LIN {X 0,Y 208.823,Z 674.449,A -85,B 0,C 180,E1 -21153.863,E2 -21153.863} C_VEL
LIN {X 0,Y 207.998,Z 678.952,A -85,B 0,C 180,E1 -21156.795,E2 -21156.795} C_VEL
LIN {X 0,Y 207.528,Z 682.383,A -85,B 0,C 180,E1 -21159.752,E2 -21159.752} C_VEL
LIN {X 0,Y 207.417,Z 684.105,A -85,B 0,C 180,E1 -21161.733,E2 -21161.733} C_VEL
LIN {X 0,Y 207.417,Z 685.435,A -85,B 0,C 180,E1 -21163.724,E2 -21163.724} C_VEL
LIN {X 0,Y 207.605,Z 686.333,A -85,B 0,C 180,E1 -21165.716,E2 -21165.716} C_VEL
LIN {X 0,Y 208.504,Z 686.886,A -85,B 0,C 180,E1 -21169.702,E2 -21169.702} C_VEL
LIN {X 0,Y 209.212,Z 686.573,A -85,B 0,C 180,E1 -21171.689,E2 -21171.689} C_VEL
LIN {X 0,Y 210.098,Z 685.804,A -85,B 0,C 180,E1 -21173.67,E2 -21173.67} C_VEL
LIN {X 0,Y 211.584,Z 684.174,A -85,B 0,C 180,E1 -21176.257,E2 -21176.257} C_VEL
LIN {X 0,Y 213.864,Z 680.916,A -85,B 0,C 180,E1 -21179.537,E2 -21179.537} C_VEL
LIN {X 0,Y 216.359,Z 676.881,A -85,B 0,C 180,E1 -21182.377,E2 -21182.377} C_VEL
LIN {X 0,Y 219.278,Z 671.481,A -85,B 0,C 180,E1 -21185.237,E2 -21185.237} C_VEL
LIN {X 0,Y 222.734,Z 664.359,A -85,B 0,C 180,E1 -21188.121,E2 -21188.121} C_VEL
LIN {X 0,Y 226.294,Z 656.011,A -85,B 0,C 180,E1 -21190.711,E2 -21190.711} C_VEL
LIN {X 0,Y 229.453,Z 647.343,A -85,B 0,C 180,E1 -21192.851,E2 -21192.851} C_VEL
LIN {X 0,Y 232.75,Z 636.876,A -85,B 0,C 180,E1 -21194.899,E2 -21194.899} C_VEL
LIN {X 0,Y 235.49,Z 626.613,A -85,B 0,C 180,E1 -21196.459,E2 -21196.459} C_VEL
LIN {X 0,Y 237.985,Z 614.319,A -85,B 0,C 180,E1 -21197.929,E2 -21197.929} C_VEL
LIN {X 0,Y 238.322,Z 612.312,A -85,B 0,C 180,E1 -21198.142,E2 -21198.142} C_VEL
LIN {X 0,Y 233.556,Z 615.33,A -85,B 0,C 180,E1 -21198.792,E2 -21198.792} C_VEL
LIN {X 0,Y 232.873,Z 615.574,A -85,B 0,C 180,E1 -21198.917,E2 -21198.917} C_VEL
LIN {X 0,Y 228.743,Z 619.885,A -85,B 0,C 180,E1 -21199.24,E2 -21199.24} C_VEL
LIN {X 0,Y 225.248,Z 622.285,A -85,B 0,C 180,E1 -21199.699,E2 -21199.699} C_VEL
LIN {X 0,Y 223.173,Z 622.996,A -85,B 0,C 180,E1 -21200.11,E2 -21200.11} C_VEL
LIN {X 0,Y 220.737,Z 624.617,A -85,B 0,C 180,E1 -21200.449,E2 -21200.449} C_VEL
LIN {X 0,Y 218.711,Z 626.309,A -85,B 0,C 180,E1 -21200.666,E2 -21200.666} C_VEL
LIN {X 0,Y 217.399,Z 627.014,A -85,B 0,C 180,E1 -21200.888,E2 -21200.888} C_VEL
LIN {X 0,Y 215.398,Z 627.078,A -85,B 0,C 180,E1 -21201.466,E2 -21201.466} C_VEL
LIN {X 0,Y 214.764,Z 627.721,A -85,B 0,C 180,E1 -21201.855,E2 -21201.855} C_VEL
LIN {X 0,Y 214.34,Z 629.899,A -85,B 0,C 180,E1 -21202.213,E2 -21202.213} C_VEL
LIN {X 0,Y 213.369,Z 648.073,A -85,B 0,C 180,E1 -21203.272,E2 -21203.272} C_VEL
LIN {X 0,Y 212.299,Z 661.771,A -85,B 0,C 180,E1 -21204.452,E2 -21204.452} C_VEL
LIN {X 0,Y 211.049,Z 675.35,A -85,B 0,C 180,E1 -21206.054,E2 -21206.054} C_VEL
LIN {X 0,Y 209.703,Z 687.117,A -85,B 0,C 180,E1 -21207.858,E2 -21207.858} C_VEL
LIN {X 0,Y 208.34,Z 699.065,A -85,B 0,C 180,E1 -21210.162,E2 -21210.162} C_VEL
LIN {X 0,Y 207.069,Z 709.634,A -85,B 0,C 180,E1 -21212.73,E2 -21212.73} C_VEL
LIN {X 0,Y 206.085,Z 718.236,A -85,B 0,C 180,E1 -21215.308,E2 -21215.308} C_VEL
LIN {X 0,Y 205.251,Z 726.508,A -85,B 0,C 180,E1 -21218.403,E2 -21218.403} C_VEL
LIN {X 0,Y 204.782,Z 732.079,A -85,B 0,C 180,E1 -21220.973,E2 -21220.973} C_VEL
LIN {X 0,Y 204.444,Z 737.792,A -85,B 0,C 180,E1 -21224.276,E2 -21224.276} C_VEL
LIN {X 0,Y 204.435,Z 741.499,A -85,B 0,C 180,E1 -21227.089,E2 -21227.089} C_VEL
LIN {X 0,Y 204.68,Z 744.43,A -85,B 0,C 180,E1 -21230.115,E2 -21230.115} C_VEL
LIN {X 0,Y 205.369,Z 746.263,A -85,B 0,C 180,E1 -21232.963,E2 -21232.963} C_VEL
LIN {X 0,Y 206.422,Z 747.309,A -85,B 0,C 180,E1 -21236.096,E2 -21236.096} C_VEL
LIN {X 0,Y 207.37,Z 747.452,A -85,B 0,C 180,E1 -21238.059,E2 -21238.059} C_VEL
LIN {X 0,Y 208.563,Z 747.149,A -85,B 0,C 180,E1 -21240.001,E2 -21240.001} C_VEL
LIN {X 0,Y 211.574,Z 745.345,A -85,B 0,C 180,E1 -21243.81,E2 -21243.81} C_VEL
LIN {X 0,Y 214.394,Z 742.884,A -85,B 0,C 180,E1 -21246.589,E2 -21246.589} C_VEL
LIN {X 0,Y 217.772,Z 739.421,A -85,B 0,C 180,E1 -21249.287,E2 -21249.287} C_VEL
LIN {X 0,Y 221.662,Z 734.872,A -85,B 0,C 180,E1 -21251.894,E2 -21251.894} C_VEL
LIN {X 0,Y 225.939,Z 729.122,A -85,B 0,C 180,E1 -21254.41,E2 -21254.41} C_VEL
LIN {X 0,Y 230.689,Z 722.012,A -85,B 0,C 180,E1 -21256.824,E2 -21256.824} C_VEL
LIN {X 0,Y 235.347,Z 714.147,A -85,B 0,C 180,E1 -21258.921,E2 -21258.921} C_VEL
LIN {X 0,Y 236.362,Z 711.674,A -85,B 0,C 180,E1 -21259.645,E2 -21259.645} C_VEL
LIN {X 0,Y 237.309,Z 704.472,A -85,B 0,C 180,E1 -21262.404,E2 -21262.404} C_VEL
LIN {X 0,Y 238.382,Z 701.707,A -85,B 0,C 180,E1 -21263.039,E2 -21263.039} C_VEL
LIN {X 0,Y 242.989,Z 691.682,A -85,B 0,C 180,E1 -21264.568,E2 -21264.568} C_VEL
LIN {X 0,Y 247.37,Z 680.576,A -85,B 0,C 180,E1 -21265.902,E2 -21265.902} C_VEL
LIN {X 0,Y 251.244,Z 668.567,A -85,B 0,C 180,E1 -21267.037,E2 -21267.037} C_VEL
LIN {X 0,Y 254.503,Z 655.536,A -85,B 0,C 180,E1 -21267.943,E2 -21267.943} C_VEL
LIN {X 0,Y 257.403,Z 640.155,A -85,B 0,C 180,E1 -21268.694,E2 -21268.694} C_VEL
LIN {X 0,Y 265.589,Z 594.222,A -85,B 0,C 180,E1 -21270.603,E2 -21270.603} C_VEL
LIN {X 0,Y 264.661,Z 590.541,A -85,B 0,C 180,E1 -21272.277,E2 -21272.277} C_VEL
LIN {X 0,Y 263.938,Z 587.985,A -85,B 0,C 180,E1 -21273.878,E2 -21273.878} C_VEL
LIN {X 0,Y 263.306,Z 585.888,A -85,B 0,C 180,E1 -21276.124,E2 -21276.124} C_VEL
LIN {X 0,Y 263.166,Z 585.155,A -85,B 0,C 180,E1 -21277.897,E2 -21277.897} C_VEL
LIN {X 0,Y 263.815,Z 585.417,A -85,B 0,C 180,E1 -21280.995,E2 -21280.995} C_VEL
LIN {X 0,Y 264.727,Z 586.842,A -85,B 0,C 180,E1 -21282.989,E2 -21282.989} C_VEL
LIN {X 0,Y 264.815,Z 590.292,A -85,B 0,C 180,E1 -21283.934,E2 -21283.934} C_VEL
LIN {X 0,Y 263.077,Z 604.973,A -85,B 0,C 180,E1 -21285.508,E2 -21285.508} C_VEL
LIN {X 0,Y 261.762,Z 615.581,A -85,B 0,C 180,E1 -21286.386,E2 -21286.386} C_VEL
LIN {X 0,Y 260.777,Z 622.254,A -85,B 0,C 180,E1 -21286.813,E2 -21286.813} C_VEL
LIN {X 0,Y 253.305,Z 663.727,A -85,B 0,C 180,E1 -21288.605,E2 -21288.605} C_VEL
LIN {X 0,Y 249.816,Z 677.135,A -85,B 0,C 180,E1 -21289.357,E2 -21289.357} C_VEL
LIN {X 0,Y 245.343,Z 690.467,A -85,B 0,C 180,E1 -21290.401,E2 -21290.401} C_VEL
LIN {X 0,Y 240.024,Z 703.488,A -85,B 0,C 180,E1 -21291.787,E2 -21291.787} C_VEL
LIN {X 0,Y 234.94,Z 714.211,A -85,B 0,C 180,E1 -21293.25,E2 -21293.25} C_VEL
LIN {X 0,Y 229.779,Z 723.994,A -85,B 0,C 180,E1 -21295.003,E2 -21295.003} C_VEL
LIN {X 0,Y 223.968,Z 733.685,A -85,B 0,C 180,E1 -21297.225,E2 -21297.225} C_VEL
LIN {X 0,Y 218.604,Z 741.763,A -85,B 0,C 180,E1 -21299.576,E2 -21299.576} C_VEL
LIN {X 0,Y 213.11,Z 749.349,A -85,B 0,C 180,E1 -21302.5,E2 -21302.5} C_VEL
LIN {X 0,Y 208.602,Z 755.144,A -85,B 0,C 180,E1 -21305.459,E2 -21305.459} C_VEL
LIN {X 0,Y 204.659,Z 759.964,A -85,B 0,C 180,E1 -21308.861,E2 -21308.861} C_VEL
LIN {X 0,Y 202.062,Z 762.893,A -85,B 0,C 180,E1 -21311.755,E2 -21311.755} C_VEL
LIN {X 0,Y 199.407,Z 765.445,A -85,B 0,C 180,E1 -21315.714,E2 -21315.714} C_VEL
LIN {X 0,Y 198.054,Z 766.417,A -85,B 0,C 180,E1 -21319.777,E2 -21319.777} C_VEL
LIN {X 0,Y 197.633,Z 765.874,A -85,B 0,C 180,E1 -21323.873,E2 -21323.873} C_VEL
LIN {X 0,Y 197.722,Z 765.004,A -85,B 0,C 180,E1 -21325.92,E2 -21325.92} C_VEL
LIN {X 0,Y 197.958,Z 763.693,A -85,B 0,C 180,E1 -21327.962,E2 -21327.962} C_VEL
LIN {X 0,Y 198.364,Z 761.941,A -85,B 0,C 180,E1 -21329.997,E2 -21329.997} C_VEL
LIN {X 0,Y 198.186,Z 758.235,A -85,B 0,C 180,E1 -21333.046,E2 -21333.046} C_VEL
LIN {X 0,Y 198.215,Z 753.277,A -85,B 0,C 180,E1 -21336.103,E2 -21336.103} C_VEL
LIN {X 0,Y 198.379,Z 746.848,A -85,B 0,C 180,E1 -21339.17,E2 -21339.17} C_VEL
LIN {X 0,Y 198.905,Z 738.692,A -85,B 0,C 180,E1 -21342.236,E2 -21342.236} C_VEL
LIN {X 0,Y 199.65,Z 730.322,A -85,B 0,C 180,E1 -21344.782,E2 -21344.782} C_VEL
LIN {X 0,Y 200.643,Z 721.169,A -85,B 0,C 180,E1 -21347.055,E2 -21347.055} C_VEL
LIN {X 0,Y 201.826,Z 711.705,A -85,B 0,C 180,E1 -21349.05,E2 -21349.05} C_VEL
LIN {X 0,Y 203.507,Z 702.102,A -85,B 0,C 180,E1 -21351.735,E2 -21351.735} C_VEL
LIN {X 0,Y 205.367,Z 692.068,A -85,B 0,C 180,E1 -21353.974,E2 -21353.974} C_VEL
LIN {X 0,Y 207.591,Z 681.441,A -85,B 0,C 180,E1 -21355.838,E2 -21355.838} C_VEL
LIN {X 0,Y 209.251,Z 671.475,A -85,B 0,C 180,E1 -21357.229,E2 -21357.229} C_VEL
LIN {X 0,Y 210.974,Z 659.917,A -85,B 0,C 180,E1 -21358.471,E2 -21358.471} C_VEL
LIN {X 0,Y 212.352,Z 646.621,A -85,B 0,C 180,E1 -21359.488,E2 -21359.488} C_VEL
LIN {X 0,Y 213.188,Z 633.325,A -85,B 0,C 180,E1 -21360.129,E2 -21360.129} C_VEL
LIN {X 0,Y 213.879,Z 609.163,A -85,B 0,C 180,E1 -21360.936,E2 -21360.936} C_VEL
LIN {X 0,Y 209.567,Z 547.865,A -85,B 0,C 180,E1 -21363.79,E2 -21363.79} C_VEL
LIN {X 0,Y 208.199,Z 533.575,A -85,B 0,C 180,E1 -21364.526,E2 -21364.526} C_VEL
LIN {X 0,Y 205.98,Z 527.108,A -85,B 0,C 180,E1 -21365.161,E2 -21365.161} C_VEL
LIN {X 0,Y 203.635,Z 515.93,A -85,B 0,C 180,E1 -21369.33,E2 -21369.33} C_VEL
LIN {X 0,Y 201.205,Z 505.753,A -85,B 0,C 180,E1 -21373.441,E2 -21373.441} C_VEL
LIN {X 0,Y 199.618,Z 499.708,A -85,B 0,C 180,E1 -21376.154,E2 -21376.154} C_VEL
LIN {X 0,Y 199.601,Z 499.613,A -85,B 0,C 180,E1 -21380.765,E2 -21380.765} C_VEL
LIN {X 0,Y 199.602,Z 499.606,A -85,B 0,C 180,E1 -21385.711,E2 -21385.711} C_VEL
LIN {X 0,Y 199.684,Z 499.613,A -85,B 0,C 180,E1 -21388.133,E2 -21388.133} C_VEL
LIN {X 0,Y 199.675,Z 499.591,A -85,B 0,C 180,E1 -21392.769,E2 -21392.769} C_VEL
LIN {X 0,Y 199.728,Z 499.604,A -85,B 0,C 180,E1 -21397.227,E2 -21397.227} C_VEL
LIN {X 0,Y 199.786,Z 499.587,A -85,B 0,C 180,E1 -21401.756,E2 -21401.756} C_VEL
LIN {X 0,Y 199.837,Z 499.591,A -85,B 0,C 180,E1 -21405.748,E2 -21405.748} C_VEL
LIN {X 0,Y 200.059,Z 499.543,A -85,B 0,C 180,E1 -21409.883,E2 -21409.883} C_VEL
LIN {X 0,Y 200.025,Z 499.568,A -85,B 0,C 180,E1 -21413.949,E2 -21413.949} C_VEL
LIN {X 0,Y 200.309,Z 499.507,A -85,B 0,C 180,E1 -21417.989,E2 -21417.989} C_VEL
LIN {X 0,Y 200.467,Z 499.492,A -85,B 0,C 180,E1 -21419.999,E2 -21419.999} C_VEL
LIN {X 0,Y 200.019,Z 499.568,A -85,B 0,C 180,E1 -21424.029,E2 -21424.029} C_VEL
LIN {X 0,Y 200.099,Z 499.533,A -85,B 0,C 180,E1 -21428.075,E2 -21428.075} C_VEL
LIN {X 0,Y 199.901,Z 499.577,A -85,B 0,C 180,E1 -21432.177,E2 -21432.177} C_VEL
LIN {X 0,Y 199.792,Z 499.59,A -85,B 0,C 180,E1 -21436.344,E2 -21436.344} C_VEL
LIN {X 0,Y 199.687,Z 499.588,A -85,B 0,C 180,E1 -21440.606,E2 -21440.606} C_VEL
LIN {X 0,Y 199.661,Z 499.612,A -85,B 0,C 180,E1 -21444.985,E2 -21444.985} C_VEL
LIN {X 0,Y 199.663,Z 499.592,A -85,B 0,C 180,E1 -21449.523,E2 -21449.523} C_VEL
LIN {X 0,Y 199.666,Z 499.611,A -85,B 0,C 180,E1 -21452.36,E2 -21452.36} C_VEL
LIN {X 0,Y 199.612,Z 499.602,A -85,B 0,C 180,E1 -21456.765,E2 -21456.765} C_VEL
LIN {X 0,Y 199.601,Z 499.613,A -85,B 0,C 180,E1 -21459.329,E2 -21459.329} C_VEL
LIN {X 0,Y 199.586,Z 499.623,A -85,B 0,C 180,E1 -21462.319,E2 -21462.319} C_VEL
LIN {X 0,Y 199.635,Z 499.603,A -85,B 0,C 180,E1 -21465.25,E2 -21465.25} C_VEL
LIN {X 0,Y 199.658,Z 499.615,A -85,B 0,C 180,E1 -21468.03,E2 -21468.03} C_VEL
LIN {X 0,Y 199.692,Z 499.59,A -85,B 0,C 180,E1 -21470.738,E2 -21470.738} C_VEL
LIN {X 0,Y 199.626,Z 499.587,A -85,B 0,C 180,E1 -21475.721,E2 -21475.721} C_VEL
LIN {X 0,Y 199.696,Z 499.611,A -85,B 0,C 180,E1 -21478.141,E2 -21478.141} C_VEL
LIN {X 0,Y 199.679,Z 499.581,A -85,B 0,C 180,E1 -21482.775,E2 -21482.775} C_VEL
LIN {X 0,Y 199.732,Z 499.589,A -85,B 0,C 180,E1 -21487.232,E2 -21487.232} C_VEL
LIN {X 0,Y 199.774,Z 499.879,A -85,B 0,C 180,E1 -21488.935,E2 -21488.935} C_VEL
LIN {X 0,Y 200.104,Z 501.145,A -85,B 0,C 180,E1 -21489.266,E2 -21489.266} C_VEL
LIN {X 0,Y 208.067,Z 516.252,A -85,B 0,C 180,E1 -21491.146,E2 -21491.146} C_VEL
LIN {X 0,Y 215.451,Z 533.098,A -85,B 0,C 180,E1 -21492.837,E2 -21492.837} C_VEL
LIN {X 0,Y 216.008,Z 534.854,A -85,B 0,C 180,E1 -21492.976,E2 -21492.976} C_VEL
LIN {X 0,Y 215.011,Z 572.79,A -85,B 0,C 180,E1 -21494.245,E2 -21494.245} C_VEL
LIN {X 0,Y 214.714,Z 587.849,A -85,B 0,C 180,E1 -21494.884,E2 -21494.884} C_VEL
LIN {X 0,Y 213.985,Z 600.276,A -85,B 0,C 180,E1 -21495.743,E2 -21495.743} C_VEL
LIN {X 0,Y 212.984,Z 611.844,A -85,B 0,C 180,E1 -21496.891,E2 -21496.891} C_VEL
LIN {X 0,Y 211.527,Z 624.08,A -85,B 0,C 180,E1 -21498.504,E2 -21498.504} C_VEL
LIN {X 0,Y 209.79,Z 635.088,A -85,B 0,C 180,E1 -21500.361,E2 -21500.361} C_VEL
LIN {X 0,Y 208.271,Z 643.991,A -85,B 0,C 180,E1 -21502.246,E2 -21502.246} C_VEL
LIN {X 0,Y 206.474,Z 653.171,A -85,B 0,C 180,E1 -21504.632,E2 -21504.632} C_VEL
LIN {X 0,Y 204.639,Z 662.104,A -85,B 0,C 180,E1 -21507.543,E2 -21507.543} C_VEL
LIN {X 0,Y 203.088,Z 669.333,A -85,B 0,C 180,E1 -21510.499,E2 -21510.499} C_VEL
LIN {X 0,Y 202.063,Z 674.223,A -85,B 0,C 180,E1 -21512.994,E2 -21512.994} C_VEL
LIN {X 0,Y 201.14,Z 678.999,A -85,B 0,C 180,E1 -21516.02,E2 -21516.02} C_VEL
LIN {X 0,Y 200.566,Z 682.673,A -85,B 0,C 180,E1 -21519.076,E2 -21519.076} C_VEL
LIN {X 0,Y 200.365,Z 685.333,A -85,B 0,C 180,E1 -21522.152,E2 -21522.152} C_VEL
LIN {X 0,Y 200.412,Z 686.599,A -85,B 0,C 180,E1 -21524.213,E2 -21524.213} C_VEL
LIN {X 0,Y 201.08,Z 687.836,A -85,B 0,C 180,E1 -21528.338,E2 -21528.338} C_VEL
LIN {X 0,Y 201.676,Z 687.872,A -85,B 0,C 180,E1 -21530.398,E2 -21530.398} C_VEL
LIN {X 0,Y 202.461,Z 687.473,A -85,B 0,C 180,E1 -21532.451,E2 -21532.451} C_VEL
LIN {X 0,Y 203.441,Z 686.643,A -85,B 0,C 180,E1 -21534.494,E2 -21534.494} C_VEL
LIN {X 0,Y 204.878,Z 685.145,A -85,B 0,C 180,E1 -21536.89,E2 -21536.89} C_VEL
LIN {X 0,Y 207.538,Z 681.544,A -85,B 0,C 180,E1 -21540.531,E2 -21540.531} C_VEL
LIN {X 0,Y 210.345,Z 677.172,A -85,B 0,C 180,E1 -21543.581,E2 -21543.581} C_VEL
LIN {X 0,Y 213.354,Z 671.867,A -85,B 0,C 180,E1 -21546.369,E2 -21546.369} C_VEL
LIN {X 0,Y 216.841,Z 664.93,A -85,B 0,C 180,E1 -21549.191,E2 -21549.191} C_VEL
LIN {X 0,Y 220.099,Z 657.662,A -85,B 0,C 180,E1 -21551.5,E2 -21551.5} C_VEL
LIN {X 0,Y 223.529,Z 648.75,A -85,B 0,C 180,E1 -21553.769,E2 -21553.769} C_VEL
LIN {X 0,Y 226.827,Z 638.829,A -85,B 0,C 180,E1 -21555.77,E2 -21555.77} C_VEL
LIN {X 0,Y 229.852,Z 628.108,A -85,B 0,C 180,E1 -21557.465,E2 -21557.465} C_VEL
LIN {X 0,Y 230.725,Z 624.603,A -85,B 0,C 180,E1 -21557.924,E2 -21557.924} C_VEL
LIN {X 0,Y 227.311,Z 626.757,A -85,B 0,C 180,E1 -21558.339,E2 -21558.339} C_VEL
LIN {X 0,Y 222.589,Z 629.079,A -85,B 0,C 180,E1 -21559.069,E2 -21559.069} C_VEL
LIN {X 0,Y 218.949,Z 631.678,A -85,B 0,C 180,E1 -21559.459,E2 -21559.459} C_VEL
LIN {X 0,Y 217.344,Z 632.498,A -85,B 0,C 180,E1 -21559.706,E2 -21559.706} C_VEL
LIN {X 0,Y 214.647,Z 633.226,A -85,B 0,C 180,E1 -21560.288,E2 -21560.288} C_VEL
LIN {X 0,Y 211.053,Z 635.602,A -85,B 0,C 180,E1 -21560.752,E2 -21560.752} C_VEL
LIN {X 0,Y 208.438,Z 636.331,A -85,B 0,C 180,E1 -21561.356,E2 -21561.356} C_VEL
LIN {X 0,Y 207.395,Z 636.47,A -85,B 0,C 180,E1 -21561.837,E2 -21561.837} C_VEL
LIN {X 0,Y 206.94,Z 638.011,A -85,B 0,C 180,E1 -21562.253,E2 -21562.253} C_VEL
LIN {X 0,Y 205.731,Z 655.76,A -85,B 0,C 180,E1 -21563.592,E2 -21563.592} C_VEL
LIN {X 0,Y 204.635,Z 668.77,A -85,B 0,C 180,E1 -21564.972,E2 -21564.972} C_VEL
LIN {X 0,Y 203.307,Z 681.341,A -85,B 0,C 180,E1 -21566.718,E2 -21566.718} C_VEL
LIN {X 0,Y 201.931,Z 693.13,A -85,B 0,C 180,E1 -21568.822,E2 -21568.822} C_VEL
LIN {X 0,Y 200.658,Z 703.559,A -85,B 0,C 180,E1 -21571.124,E2 -21571.124} C_VEL
LIN {X 0,Y 199.491,Z 713.576,A -85,B 0,C 180,E1 -21573.873,E2 -21573.873} C_VEL
LIN {X 0,Y 198.616,Z 721.694,A -85,B 0,C 180,E1 -21576.598,E2 -21576.598} C_VEL
LIN {X 0,Y 197.914,Z 729.243,A -85,B 0,C 180,E1 -21579.744,E2 -21579.744} C_VEL
LIN {X 0,Y 197.544,Z 734.412,A -85,B 0,C 180,E1 -21582.399,E2 -21582.399} C_VEL
LIN {X 0,Y 197.318,Z 739.285,A -85,B 0,C 180,E1 -21585.563,E2 -21585.563} C_VEL
LIN {X 0,Y 197.395,Z 742.957,A -85,B 0,C 180,E1 -21588.708,E2 -21588.708} C_VEL
LIN {X 0,Y 198.265,Z 746.338,A -85,B 0,C 180,E1 -21593.016,E2 -21593.016} C_VEL
LIN {X 0,Y 199.254,Z 747.581,A -85,B 0,C 180,E1 -21595.956,E2 -21595.956} C_VEL
LIN {X 0,Y 200.172,Z 747.933,A -85,B 0,C 180,E1 -21597.989,E2 -21597.989} C_VEL
LIN {X 0,Y 202.8,Z 747.429,A -85,B 0,C 180,E1 -21601.987,E2 -21601.987} C_VEL
LIN {X 0,Y 204.442,Z 746.584,A -85,B 0,C 180,E1 -21603.943,E2 -21603.943} C_VEL
LIN {X 0,Y 208.453,Z 743.607,A -85,B 0,C 180,E1 -21607.751,E2 -21607.751} C_VEL
LIN {X 0,Y 212.086,Z 740.232,A -85,B 0,C 180,E1 -21610.502,E2 -21610.502} C_VEL
LIN {X 0,Y 216.856,Z 735.067,A -85,B 0,C 180,E1 -21613.517,E2 -21613.517} C_VEL
LIN {X 0,Y 221.641,Z 729.115,A -85,B 0,C 180,E1 -21616.109,E2 -21616.109} C_VEL
LIN {X 0,Y 226.784,Z 721.829,A -85,B 0,C 180,E1 -21618.521,E2 -21618.521} C_VEL
LIN {X 0,Y 232.326,Z 712.998,A -85,B 0,C 180,E1 -21620.821,E2 -21620.821} C_VEL
LIN {X 0,Y 237.753,Z 702.943,A -85,B 0,C 180,E1 -21622.828,E2 -21622.828} C_VEL
LIN {X 0,Y 238.382,Z 701.707,A -85,B 0,C 180,E1 -21623.039,E2 -21623.039} C_VEL
LIN {X 0,Y 240.262,Z 697.383,A -85,B 0,C 180,E1 -21623.893,E2 -21623.893} C_VEL
LIN {X 0,Y 242.264,Z 690.529,A -85,B 0,C 180,E1 -21625.528,E2 -21625.528} C_VEL
LIN {X 0,Y 244.08,Z 683.301,A -85,B 0,C 180,E1 -21627.049,E2 -21627.049} C_VEL
LIN {X 0,Y 245.594,Z 678.404,A -85,B 0,C 180,E1 -21627.719,E2 -21627.719} C_VEL
LIN {X 0,Y 249.586,Z 666.071,A -85,B 0,C 180,E1 -21628.802,E2 -21628.802} C_VEL
LIN {X 0,Y 252.788,Z 653.392,A -85,B 0,C 180,E1 -21629.622,E2 -21629.622} C_VEL
LIN {X 0,Y 261.13,Z 609.162,A -85,B 0,C 180,E1 -21631.487,E2 -21631.487} C_VEL
LIN {X 0,Y 263.114,Z 598.685,A -85,B 0,C 180,E1 -21631.925,E2 -21631.925} C_VEL
LIN {X 0,Y 262.323,Z 595.278,A -85,B 0,C 180,E1 -21633.792,E2 -21633.792} C_VEL
LIN {X 0,Y 261.743,Z 592.897,A -85,B 0,C 180,E1 -21636.031,E2 -21636.031} C_VEL
LIN {X 0,Y 261.593,Z 592.046,A -85,B 0,C 180,E1 -21638.165,E2 -21638.165} C_VEL
LIN {X 0,Y 262.204,Z 592.337,A -85,B 0,C 180,E1 -21640.917,E2 -21640.917} C_VEL
LIN {X 0,Y 262.837,Z 593.531,A -85,B 0,C 180,E1 -21642.467,E2 -21642.467} C_VEL
LIN {X 0,Y 262.757,Z 594.797,A -85,B 0,C 180,E1 -21642.782,E2 -21642.782} C_VEL
LIN {X 0,Y 260.745,Z 609.605,A -85,B 0,C 180,E1 -21644.334,E2 -21644.334} C_VEL
LIN {X 0,Y 258.929,Z 621.439,A -85,B 0,C 180,E1 -21645.255,E2 -21645.255} C_VEL
LIN {X 0,Y 251.215,Z 662.471,A -85,B 0,C 180,E1 -21647.003,E2 -21647.003} C_VEL
LIN {X 0,Y 247.446,Z 676.313,A -85,B 0,C 180,E1 -21647.77,E2 -21647.77} C_VEL
LIN {X 0,Y 243.339,Z 688.05,A -85,B 0,C 180,E1 -21648.646,E2 -21648.646} C_VEL
LIN {X 0,Y 238.399,Z 700.138,A -85,B 0,C 180,E1 -21649.84,E2 -21649.84} C_VEL
LIN {X 0,Y 232.961,Z 711.254,A -85,B 0,C 180,E1 -21651.242,E2 -21651.242} C_VEL
LIN {X 0,Y 227.353,Z 721.318,A -85,B 0,C 180,E1 -21652.927,E2 -21652.927} C_VEL
LIN {X 0,Y 221.136,Z 731.437,A -85,B 0,C 180,E1 -21655.102,E2 -21655.102} C_VEL
LIN {X 0,Y 215.337,Z 739.681,A -85,B 0,C 180,E1 -21657.414,E2 -21657.414} C_VEL
LIN {X 0,Y 209.296,Z 747.575,A -85,B 0,C 180,E1 -21660.307,E2 -21660.307} C_VEL
LIN {X 0,Y 205.477,Z 752.177,A -85,B 0,C 180,E1 -21662.497,E2 -21662.497} C_VEL
LIN {X 0,Y 200.5,Z 757.664,A -85,B 0,C 180,E1 -21665.894,E2 -21665.894} C_VEL
LIN {X 0,Y 197.086,Z 761.314,A -85,B 0,C 180,E1 -21669.105,E2 -21669.105} C_VEL
LIN {X 0,Y 195.334,Z 762.996,A -85,B 0,C 180,E1 -21671.103,E2 -21671.103} C_VEL
LIN {X 0,Y 192.502,Z 765.193,A -85,B 0,C 180,E1 -21675.19,E2 -21675.19} C_VEL
LIN {X 0,Y 191.037,Z 765.925,A -85,B 0,C 180,E1 -21679.397,E2 -21679.397} C_VEL
LIN {X 0,Y 190.664,Z 765.714,A -85,B 0,C 180,E1 -21681.518,E2 -21681.518} C_VEL
LIN {X 0,Y 190.681,Z 764.073,A -85,B 0,C 180,E1 -21685.769,E2 -21685.769} C_VEL
LIN {X 0,Y 190.942,Z 762.656,A -85,B 0,C 180,E1 -21687.887,E2 -21687.887} C_VEL
LIN {X 0,Y 191.341,Z 760.803,A -85,B 0,C 180,E1 -21689.996,E2 -21689.996} C_VEL
LIN {X 0,Y 191.178,Z 756.892,A -85,B 0,C 180,E1 -21693.157,E2 -21693.157} C_VEL
LIN {X 0,Y 191.209,Z 751.637,A -85,B 0,C 180,E1 -21696.327,E2 -21696.327} C_VEL
LIN {X 0,Y 191.415,Z 744.881,A -85,B 0,C 180,E1 -21699.506,E2 -21699.506} C_VEL
LIN {X 0,Y 191.963,Z 736.355,A -85,B 0,C 180,E1 -21702.686,E2 -21702.686} C_VEL
LIN {X 0,Y 192.847,Z 727.556,A -85,B 0,C 180,E1 -21705.317,E2 -21705.317} C_VEL
LIN {X 0,Y 194.076,Z 716.807,A -85,B 0,C 180,E1 -21707.923,E2 -21707.923} C_VEL
LIN {X 0,Y 194.48,Z 713.213,A -85,B 0,C 180,E1 -21708.703,E2 -21708.703} C_VEL
LIN {X 0,Y 196.118,Z 704.192,A -85,B 0,C 180,E1 -21711.491,E2 -21711.491} C_VEL
LIN {X 0,Y 198.146,Z 693.75,A -85,B 0,C 180,E1 -21714.068,E2 -21714.068} C_VEL
LIN {X 0,Y 200.304,Z 683.678,A -85,B 0,C 180,E1 -21716.009,E2 -21716.009} C_VEL
LIN {X 0,Y 202.266,Z 672.677,A -85,B 0,C 180,E1 -21717.689,E2 -21717.689} C_VEL
LIN {X 0,Y 204.219,Z 660.603,A -85,B 0,C 180,E1 -21719.08,E2 -21719.08} C_VEL
LIN {X 0,Y 205.73,Z 647.377,A -85,B 0,C 180,E1 -21720.182,E2 -21720.182} C_VEL
LIN {X 0,Y 206.712,Z 633.368,A -85,B 0,C 180,E1 -21720.907,E2 -21720.907} C_VEL
LIN {X 0,Y 207.395,Z 609.475,A -85,B 0,C 180,E1 -21721.738,E2 -21721.738} C_VEL
LIN {X 0,Y 203.373,Z 549.599,A -85,B 0,C 180,E1 -21724.62,E2 -21724.62} C_VEL
LIN {X 0,Y 201.963,Z 535.388,A -85,B 0,C 180,E1 -21725.4,E2 -21725.4} C_VEL
LIN {X 0,Y 198.533,Z 525.931,A -85,B 0,C 180,E1 -21726.392,E2 -21726.392} C_VEL
LIN {X 0,Y 196.328,Z 515.452,A -85,B 0,C 180,E1 -21730.503,E2 -21730.503} C_VEL
LIN {X 0,Y 193.759,Z 504.988,A -85,B 0,C 180,E1 -21734.983,E2 -21734.983} C_VEL
LIN {X 0,Y 192.553,Z 500.605,A -85,B 0,C 180,E1 -21737.07,E2 -21737.07} C_VEL
LIN {X 0,Y 192.542,Z 500.498,A -85,B 0,C 180,E1 -21741.645,E2 -21741.645} C_VEL
LIN {X 0,Y 192.587,Z 500.487,A -85,B 0,C 180,E1 -21746.811,E2 -21746.811} C_VEL
LIN {X 0,Y 192.651,Z 500.463,A -85,B 0,C 180,E1 -21751.689,E2 -21751.689} C_VEL
LIN {X 0,Y 192.696,Z 500.484,A -85,B 0,C 180,E1 -21756.346,E2 -21756.346} C_VEL
LIN {X 0,Y 192.721,Z 500.463,A -85,B 0,C 180,E1 -21761.456,E2 -21761.456} C_VEL
LIN {X 0,Y 192.761,Z 500.472,A -85,B 0,C 180,E1 -21765.213,E2 -21765.213} C_VEL
LIN {X 0,Y 192.969,Z 500.422,A -85,B 0,C 180,E1 -21769.507,E2 -21769.507} C_VEL
LIN {X 0,Y 193.056,Z 500.43,A -85,B 0,C 180,E1 -21771.626,E2 -21771.626} C_VEL
LIN {X 0,Y 193.251,Z 500.385,A -85,B 0,C 180,E1 -21777.915,E2 -21777.915} C_VEL
LIN {X 0,Y 193.431,Z 500.367,A -85,B 0,C 180,E1 -21779.999,E2 -21779.999} C_VEL
LIN {X 0,Y 192.965,Z 500.447,A -85,B 0,C 180,E1 -21784.176,E2 -21784.176} C_VEL
LIN {X 0,Y 193.049,Z 500.408,A -85,B 0,C 180,E1 -21788.372,E2 -21788.372} C_VEL
LIN {X 0,Y 192.84,Z 500.459,A -85,B 0,C 180,E1 -21792.63,E2 -21792.63} C_VEL
LIN {X 0,Y 192.745,Z 500.463,A -85,B 0,C 180,E1 -21796.959,E2 -21796.959} C_VEL
LIN {X 0,Y 192.624,Z 500.475,A -85,B 0,C 180,E1 -21801.398,E2 -21801.398} C_VEL
LIN {X 0,Y 192.652,Z 500.486,A -85,B 0,C 180,E1 -21804.225,E2 -21804.225} C_VEL
LIN {X 0,Y 192.638,Z 500.464,A -85,B 0,C 180,E1 -21808.893,E2 -21808.893} C_VEL
LIN {X 0,Y 192.587,Z 500.496,A -85,B 0,C 180,E1 -21813.187,E2 -21813.187} C_VEL
LIN {X 0,Y 192.542,Z 500.483,A -85,B 0,C 180,E1 -21818.353,E2 -21818.353} C_VEL
LIN {X 0,Y 192.527,Z 500.495,A -85,B 0,C 180,E1 -21823.113,E2 -21823.113} C_VEL
LIN {X 0,Y 192.591,Z 500.491,A -85,B 0,C 180,E1 -21826.872,E2 -21826.872} C_VEL
LIN {X 0,Y 192.603,Z 500.455,A -85,B 0,C 180,E1 -21831.665,E2 -21831.665} C_VEL
LIN {X 0,Y 192.592,Z 500.481,A -85,B 0,C 180,E1 -21836.817,E2 -21836.817} C_VEL
LIN {X 0,Y 192.657,Z 500.454,A -85,B 0,C 180,E1 -21841.695,E2 -21841.695} C_VEL
LIN {X 0,Y 192.685,Z 500.558,A -85,B 0,C 180,E1 -21847.487,E2 -21847.487} C_VEL
LIN {X 0,Y 192.833,Z 501.316,A -85,B 0,C 180,E1 -21847.942,E2 -21847.942} C_VEL
LIN {X 0,Y 195.216,Z 506.082,A -85,B 0,C 180,E1 -21848.649,E2 -21848.649} C_VEL
LIN {X 0,Y 202.352,Z 519.518,A -85,B 0,C 180,E1 -21850.393,E2 -21850.393} C_VEL
LIN {X 0,Y 208.723,Z 534.142,A -85,B 0,C 180,E1 -21851.937,E2 -21851.937} C_VEL
LIN {X 0,Y 209.566,Z 536.101,A -85,B 0,C 180,E1 -21852.133,E2 -21852.133} C_VEL
LIN {X 0,Y 208.429,Z 583.906,A -85,B 0,C 180,E1 -21853.836,E2 -21853.836} C_VEL
LIN {X 0,Y 207.792,Z 596.77,A -85,B 0,C 180,E1 -21854.619,E2 -21854.619} C_VEL
LIN {X 0,Y 206.759,Z 610.123,A -85,B 0,C 180,E1 -21855.862,E2 -21855.862} C_VEL
LIN {X 0,Y 205.36,Z 622.257,A -85,B 0,C 180,E1 -21857.402,E2 -21857.402} C_VEL
LIN {X 0,Y 203.538,Z 633.772,A -85,B 0,C 180,E1 -21859.308,E2 -21859.308} C_VEL
LIN {X 0,Y 201.682,Z 644.139,A -85,B 0,C 180,E1 -21861.487,E2 -21861.487} C_VEL
LIN {X 0,Y 199.793,Z 653.51,A -85,B 0,C 180,E1 -21863.946,E2 -21863.946} C_VEL
LIN {X 0,Y 197.861,Z 662.549,A -85,B 0,C 180,E1 -21866.949,E2 -21866.949} C_VEL
LIN {X 0,Y 196.226,Z 669.873,A -85,B 0,C 180,E1 -21870.003,E2 -21870.003} C_VEL
LIN {X 0,Y 194.954,Z 675.76,A -85,B 0,C 180,E1 -21873.103,E2 -21873.103} C_VEL
LIN {X 0,Y 194.019,Z 680.422,A -85,B 0,C 180,E1 -21876.242,E2 -21876.242} C_VEL
LIN {X 0,Y 193.484,Z 683.99,A -85,B 0,C 180,E1 -21879.411,E2 -21879.411} C_VEL
LIN {X 0,Y 193.328,Z 686.556,A -85,B 0,C 180,E1 -21882.602,E2 -21882.602} C_VEL
LIN {X 0,Y 193.42,Z 687.728,A -85,B 0,C 180,E1 -21884.738,E2 -21884.738} C_VEL
LIN {X 0,Y 194.216,Z 688.869,A -85,B 0,C 180,E1 -21889.01,E2 -21889.01} C_VEL
LIN {X 0,Y 194.877,Z 688.839,A -85,B 0,C 180,E1 -21891.143,E2 -21891.143} C_VEL
LIN {X 0,Y 195.771,Z 688.357,A -85,B 0,C 180,E1 -21893.263,E2 -21893.263} C_VEL
LIN {X 0,Y 196.835,Z 687.481,A -85,B 0,C 180,E1 -21895.373,E2 -21895.373} C_VEL
LIN {X 0,Y 198.202,Z 686.113,A -85,B 0,C 180,E1 -21897.569,E2 -21897.569} C_VEL
LIN {X 0,Y 200.426,Z 683.375,A -85,B 0,C 180,E1 -21900.564,E2 -21900.564} C_VEL
LIN {X 0,Y 203.629,Z 678.714,A -85,B 0,C 180,E1 -21904.074,E2 -21904.074} C_VEL
LIN {X 0,Y 207.507,Z 672.254,A -85,B 0,C 180,E1 -21907.567,E2 -21907.567} C_VEL
LIN {X 0,Y 211.083,Z 665.353,A -85,B 0,C 180,E1 -21910.364,E2 -21910.364} C_VEL
LIN {X 0,Y 214.656,Z 657.666,A -85,B 0,C 180,E1 -21912.798,E2 -21912.798} C_VEL
LIN {X 0,Y 218.287,Z 648.557,A -85,B 0,C 180,E1 -21915.102,E2 -21915.102} C_VEL
LIN {X 0,Y 221.749,Z 638.365,A -85,B 0,C 180,E1 -21917.135,E2 -21917.135} C_VEL
LIN {X 0,Y 222.86,Z 634.414,A -85,B 0,C 180,E1 -21917.817,E2 -21917.817} C_VEL
LIN {X 0,Y 220.647,Z 635.907,A -85,B 0,C 180,E1 -21918.02,E2 -21918.02} C_VEL
LIN {X 0,Y 217.234,Z 637.76,A -85,B 0,C 180,E1 -21918.455,E2 -21918.455} C_VEL
LIN {X 0,Y 213.905,Z 638.828,A -85,B 0,C 180,E1 -21919.089,E2 -21919.089} C_VEL
LIN {X 0,Y 210.788,Z 640.793,A -85,B 0,C 180,E1 -21919.446,E2 -21919.446} C_VEL
LIN {X 0,Y 207.88,Z 641.724,A -85,B 0,C 180,E1 -21920.034,E2 -21920.034} C_VEL
LIN {X 0,Y 201.843,Z 644.118,A -85,B 0,C 180,E1 -21921.191,E2 -21921.191} C_VEL
LIN {X 0,Y 199.983,Z 644.138,A -85,B 0,C 180,E1 -21921.969,E2 -21921.969} C_VEL
LIN {X 0,Y 199.521,Z 645.568,A -85,B 0,C 180,E1 -21922.424,E2 -21922.424} C_VEL
LIN {X 0,Y 198.219,Z 661.925,A -85,B 0,C 180,E1 -21923.952,E2 -21923.952} C_VEL
LIN {X 0,Y 196.813,Z 676.322,A -85,B 0,C 180,E1 -21925.778,E2 -21925.778} C_VEL
LIN {X 0,Y 195.314,Z 689.235,A -85,B 0,C 180,E1 -21927.945,E2 -21927.945} C_VEL
LIN {X 0,Y 193.893,Z 700.999,A -85,B 0,C 180,E1 -21930.456,E2 -21930.456} C_VEL
LIN {X 0,Y 192.768,Z 710.228,A -85,B 0,C 180,E1 -21932.889,E2 -21932.889} C_VEL
LIN {X 0,Y 191.784,Z 718.882,A -85,B 0,C 180,E1 -21935.654,E2 -21935.654} C_VEL
LIN {X 0,Y 190.977,Z 727.184,A -85,B 0,C 180,E1 -21938.974,E2 -21938.974} C_VEL
LIN {X 0,Y 190.528,Z 732.751,A -85,B 0,C 180,E1 -21941.728,E2 -21941.728} C_VEL
LIN {X 0,Y 190.266,Z 738.1,A -85,B 0,C 180,E1 -21945.016,E2 -21945.016} C_VEL
LIN {X 0,Y 190.287,Z 742.204,A -85,B 0,C 180,E1 -21948.28,E2 -21948.28} C_VEL
LIN {X 0,Y 190.756,Z 745.214,A -85,B 0,C 180,E1 -21951.526,E2 -21951.526} C_VEL
LIN {X 0,Y 191.337,Z 746.669,A -85,B 0,C 180,E1 -21953.674,E2 -21953.674} C_VEL
LIN {X 0,Y 192.049,Z 747.672,A -85,B 0,C 180,E1 -21955.804,E2 -21955.804} C_VEL
LIN {X 0,Y 194.197,Z 748.475,A -85,B 0,C 180,E1 -21960.001,E2 -21960.001} C_VEL
LIN {X 0,Y 195.637,Z 748.286,A -85,B 0,C 180,E1 -21962.059,E2 -21962.059} C_VEL
LIN {X 0,Y 199.252,Z 746.653,A -85,B 0,C 180,E1 -21966.075,E2 -21966.075} C_VEL
LIN {X 0,Y 201.423,Z 745.241,A -85,B 0,C 180,E1 -21968.024,E2 -21968.024} C_VEL
LIN {X 0,Y 205.177,Z 742.284,A -85,B 0,C 180,E1 -21970.86,E2 -21970.86} C_VEL
LIN {X 0,Y 209.947,Z 737.847,A -85,B 0,C 180,E1 -21973.874,E2 -21973.874} C_VEL
LIN {X 0,Y 215.008,Z 732.255,A -85,B 0,C 180,E1 -21976.62,E2 -21976.62} C_VEL
LIN {X 0,Y 221.233,Z 724.466,A -85,B 0,C 180,E1 -21979.486,E2 -21979.486} C_VEL
LIN {X 0,Y 226.999,Z 716.077,A -85,B 0,C 180,E1 -21981.81,E2 -21981.81} C_VEL
LIN {X 0,Y 233.212,Z 705.728,A -85,B 0,C 180,E1 -21984.007,E2 -21984.007} C_VEL
LIN {X 0,Y 238.683,Z 695.031,A -85,B 0,C 180,E1 -21985.742,E2 -21985.742} C_VEL
LIN {X 0,Y 243.25,Z 684.517,A -85,B 0,C 180,E1 -21987.069,E2 -21987.069} C_VEL
LIN {X 0,Y 245.594,Z 678.404,A -85,B 0,C 180,E1 -21987.719,E2 -21987.719} C_VEL
LIN {X 0,Y 247.134,Z 673.363,A -85,B 0,C 180,E1 -21988.353,E2 -21988.353} C_VEL
LIN {X 0,Y 248.752,Z 665.37,A -85,B 0,C 180,E1 -21989.666,E2 -21989.666} C_VEL
LIN {X 0,Y 250.209,Z 657.117,A -85,B 0,C 180,E1 -21990.845,E2 -21990.845} C_VEL
LIN {X 0,Y 251.302,Z 651.696,A -85,B 0,C 180,E1 -21991.28,E2 -21991.28} C_VEL
LIN {X 0,Y 259.606,Z 609.541,A -85,B 0,C 180,E1 -21993.012,E2 -21993.012} C_VEL
LIN {X 0,Y 260.789,Z 603.387,A -85,B 0,C 180,E1 -21993.288,E2 -21993.288} C_VEL
LIN {X 0,Y 260.322,Z 600.778,A -85,B 0,C 180,E1 -21995.097,E2 -21995.097} C_VEL
LIN {X 0,Y 260.061,Z 599.216,A -85,B 0,C 180,E1 -21997.205,E2 -21997.205} C_VEL
LIN {X 0,Y 260.049,Z 598.953,A -85,B 0,C 180,E1 -21998.433,E2 -21998.433} C_VEL
LIN {X 0,Y 260.637,Z 599.311,A -85,B 0,C 180,E1 -22000.97,E2 -22000.97} C_VEL
LIN {X 0,Y 260.914,Z 599.654,A -85,B 0,C 180,E1 -22001.618,E2 -22001.618} C_VEL
LIN {X 0,Y 258.751,Z 612.804,A -85,B 0,C 180,E1 -22002.987,E2 -22002.987} C_VEL
LIN {X 0,Y 256.964,Z 623.644,A -85,B 0,C 180,E1 -22003.806,E2 -22003.806} C_VEL
LIN {X 0,Y 249.508,Z 661.099,A -85,B 0,C 180,E1 -22005.373,E2 -22005.373} C_VEL
LIN {X 0,Y 245.076,Z 676.616,A -85,B 0,C 180,E1 -22006.21,E2 -22006.21} C_VEL
LIN {X 0,Y 240.976,Z 687.819,A -85,B 0,C 180,E1 -22007.018,E2 -22007.018} C_VEL
LIN {X 0,Y 235.48,Z 700.414,A -85,B 0,C 180,E1 -22008.258,E2 -22008.258} C_VEL
LIN {X 0,Y 229.528,Z 711.721,A -85,B 0,C 180,E1 -22009.693,E2 -22009.693} C_VEL
LIN {X 0,Y 223.088,Z 722.598,A -85,B 0,C 180,E1 -22011.52,E2 -22011.52} C_VEL
LIN {X 0,Y 216.585,Z 732.185,A -85,B 0,C 180,E1 -22013.683,E2 -22013.683} C_VEL
LIN {X 0,Y 209.531,Z 741.448,A -85,B 0,C 180,E1 -22016.394,E2 -22016.394} C_VEL
LIN {X 0,Y 204.104,Z 747.846,A -85,B 0,C 180,E1 -22018.899,E2 -22018.899} C_VEL
LIN {X 0,Y 199.273,Z 753.111,A -85,B 0,C 180,E1 -22021.564,E2 -22021.564} C_VEL
LIN {X 0,Y 193.919,Z 758.319,A -85,B 0,C 180,E1 -22025.166,E2 -22025.166} C_VEL
LIN {X 0,Y 190.453,Z 761.501,A -85,B 0,C 180,E1 -22028.341,E2 -22028.341} C_VEL
LIN {X 0,Y 186.943,Z 764.166,A -85,B 0,C 180,E1 -22032.493,E2 -22032.493} C_VEL
LIN {X 0,Y 185.615,Z 764.94,A -85,B 0,C 180,E1 -22034.627,E2 -22034.627} C_VEL
LIN {X 0,Y 184.042,Z 765.335,A -85,B 0,C 180,E1 -22038.989,E2 -22038.989} C_VEL
LIN {X 0,Y 183.549,Z 764.252,A -85,B 0,C 180,E1 -22043.4,E2 -22043.4} C_VEL
LIN {X 0,Y 183.642,Z 763.139,A -85,B 0,C 180,E1 -22045.607,E2 -22045.607} C_VEL
LIN {X 0,Y 184.097,Z 760.61,A -85,B 0,C 180,E1 -22048.903,E2 -22048.903} C_VEL
LIN {X 0,Y 184.332,Z 759.527,A -85,B 0,C 180,E1 -22049.996,E2 -22049.996} C_VEL
LIN {X 0,Y 184.189,Z 755.37,A -85,B 0,C 180,E1 -22053.277,E2 -22053.277} C_VEL
LIN {X 0,Y 184.203,Z 749.891,A -85,B 0,C 180,E1 -22056.569,E2 -22056.569} C_VEL
LIN {X 0,Y 184.46,Z 742.876,A -85,B 0,C 180,E1 -22059.868,E2 -22059.868} C_VEL
LIN {X 0,Y 185.087,Z 733.909,A -85,B 0,C 180,E1 -22063.165,E2 -22063.165} C_VEL
LIN {X 0,Y 186.047,Z 724.715,A -85,B 0,C 180,E1 -22065.891,E2 -22065.891} C_VEL
LIN {X 0,Y 187.312,Z 713.865,A -85,B 0,C 180,E1 -22068.594,E2 -22068.594} C_VEL
LIN {X 0,Y 188.953,Z 704.915,A -85,B 0,C 180,E1 -22071.585,E2 -22071.585} C_VEL
LIN {X 0,Y 191.12,Z 694.083,A -85,B 0,C 180,E1 -22074.433,E2 -22074.433} C_VEL
LIN {X 0,Y 193.308,Z 684.333,A -85,B 0,C 180,E1 -22076.443,E2 -22076.443} C_VEL
LIN {X 0,Y 195.328,Z 673.807,A -85,B 0,C 180,E1 -22078.176,E2 -22078.176} C_VEL
LIN {X 0,Y 197.307,Z 662.352,A -85,B 0,C 180,E1 -22079.614,E2 -22079.614} C_VEL
LIN {X 0,Y 198.887,Z 650.189,A -85,B 0,C 180,E1 -22080.745,E2 -22080.745} C_VEL
LIN {X 0,Y 200.052,Z 637.018,A -85,B 0,C 180,E1 -22081.574,E2 -22081.574} C_VEL
LIN {X 0,Y 200.969,Z 609.759,A -85,B 0,C 180,E1 -22082.587,E2 -22082.587} C_VEL
LIN {X 0,Y 197.079,Z 550.202,A -85,B 0,C 180,E1 -22085.57,E2 -22085.57} C_VEL
LIN {X 0,Y 195.865,Z 537.399,A -85,B 0,C 180,E1 -22086.3,E2 -22086.3} C_VEL
LIN {X 0,Y 191.12,Z 524.847,A -85,B 0,C 180,E1 -22087.704,E2 -22087.704} C_VEL
LIN {X 0,Y 188.815,Z 514.328,A -85,B 0,C 180,E1 -22092.061,E2 -22092.061} C_VEL
LIN {X 0,Y 186.46,Z 505.043,A -85,B 0,C 180,E1 -22096.297,E2 -22096.297} C_VEL
LIN {X 0,Y 185.507,Z 501.451,A -85,B 0,C 180,E1 -22098.171,E2 -22098.171} C_VEL
LIN {X 0,Y 185.498,Z 501.38,A -85,B 0,C 180,E1 -22102.708,E2 -22102.708} C_VEL
LIN {X 0,Y 185.533,Z 501.374,A -85,B 0,C 180,E1 -22107.972,E2 -22107.972} C_VEL
LIN {X 0,Y 185.571,Z 501.351,A -85,B 0,C 180,E1 -22110.574,E2 -22110.574} C_VEL
LIN {X 0,Y 185.578,Z 501.367,A -85,B 0,C 180,E1 -22115.38,E2 -22115.38} C_VEL
LIN {X 0,Y 185.664,Z 501.338,A -85,B 0,C 180,E1 -22121.131,E2 -22121.131} C_VEL
LIN {X 0,Y 185.713,Z 501.352,A -85,B 0,C 180,E1 -22124.638,E2 -22124.638} C_VEL
LIN {X 0,Y 185.913,Z 501.3,A -85,B 0,C 180,E1 -22129.357,E2 -22129.357} C_VEL
LIN {X 0,Y 185.952,Z 501.32,A -85,B 0,C 180,E1 -22133.489,E2 -22133.489} C_VEL
LIN {X 0,Y 186.195,Z 501.263,A -85,B 0,C 180,E1 -22137.836,E2 -22137.836} C_VEL
LIN {X 0,Y 186.394,Z 501.242,A -85,B 0,C 180,E1 -22139.999,E2 -22139.999} C_VEL
LIN {X 0,Y 185.913,Z 501.326,A -85,B 0,C 180,E1 -22144.335,E2 -22144.335} C_VEL
LIN {X 0,Y 185.996,Z 501.285,A -85,B 0,C 180,E1 -22148.692,E2 -22148.692} C_VEL
LIN {X 0,Y 185.752,Z 501.346,A -85,B 0,C 180,E1 -22153.12,E2 -22153.12} C_VEL
LIN {X 0,Y 185.678,Z 501.335,A -85,B 0,C 180,E1 -22157.625,E2 -22157.625} C_VEL
LIN {X 0,Y 185.584,Z 501.359,A -85,B 0,C 180,E1 -22162.252,E2 -22162.252} C_VEL
LIN {X 0,Y 185.551,Z 501.356,A -85,B 0,C 180,E1 -22167.033,E2 -22167.033} C_VEL
LIN {X 0,Y 185.567,Z 501.345,A -85,B 0,C 180,E1 -22169.494,E2 -22169.494} C_VEL
LIN {X 0,Y 185.488,Z 501.376,A -85,B 0,C 180,E1 -22174.633,E2 -22174.633} C_VEL
LIN {X 0,Y 185.495,Z 501.357,A -85,B 0,C 180,E1 -22177.315,E2 -22177.315} C_VEL
LIN {X 0,Y 185.47,Z 501.382,A -85,B 0,C 180,E1 -22180.73,E2 -22180.73} C_VEL
LIN {X 0,Y 185.544,Z 501.362,A -85,B 0,C 180,E1 -22186.027,E2 -22186.027} C_VEL
LIN {X 0,Y 185.547,Z 501.359,A -85,B 0,C 180,E1 -22189.921,E2 -22189.921} C_VEL
LIN {X 0,Y 185.566,Z 501.319,A -85,B 0,C 180,E1 -22192.706,E2 -22192.706} C_VEL
LIN {X 0,Y 185.537,Z 501.375,A -85,B 0,C 180,E1 -22197.978,E2 -22197.978} C_VEL
LIN {X 0,Y 185.574,Z 501.343,A -85,B 0,C 180,E1 -22200.579,E2 -22200.579} C_VEL
LIN {X 0,Y 185.68,Z 501.481,A -85,B 0,C 180,E1 -22206.29,E2 -22206.29} C_VEL
LIN {X 0,Y 185.864,Z 502.393,A -85,B 0,C 180,E1 -22206.703,E2 -22206.703} C_VEL
LIN {X 0,Y 196.072,Z 521.521,A -85,B 0,C 180,E1 -22209.45,E2 -22209.45} C_VEL
LIN {X 0,Y 202.453,Z 536.073,A -85,B 0,C 180,E1 -22211.076,E2 -22211.076} C_VEL
LIN {X 0,Y 203.286,Z 538.125,A -85,B 0,C 180,E1 -22211.286,E2 -22211.286} C_VEL
LIN {X 0,Y 202.085,Z 582.842,A -85,B 0,C 180,E1 -22212.904,E2 -22212.904} C_VEL
LIN {X 0,Y 201.495,Z 596.224,A -85,B 0,C 180,E1 -22213.683,E2 -22213.683} C_VEL
LIN {X 0,Y 200.542,Z 608.276,A -85,B 0,C 180,E1 -22214.765,E2 -22214.765} C_VEL
LIN {X 0,Y 199.213,Z 620.182,A -85,B 0,C 180,E1 -22216.227,E2 -22216.227} C_VEL
LIN {X 0,Y 197.341,Z 632.44,A -85,B 0,C 180,E1 -22218.187,E2 -22218.187} C_VEL
LIN {X 0,Y 195.322,Z 643.227,A -85,B 0,C 180,E1 -22220.424,E2 -22220.424} C_VEL
LIN {X 0,Y 193.512,Z 652.039,A -85,B 0,C 180,E1 -22222.701,E2 -22222.701} C_VEL
LIN {X 0,Y 191.42,Z 661.628,A -85,B 0,C 180,E1 -22225.793,E2 -22225.793} C_VEL
LIN {X 0,Y 189.8,Z 668.813,A -85,B 0,C 180,E1 -22228.724,E2 -22228.724} C_VEL
LIN {X 0,Y 188.223,Z 675.468,A -85,B 0,C 180,E1 -22232.143,E2 -22232.143} C_VEL
LIN {X 0,Y 187.172,Z 680.398,A -85,B 0,C 180,E1 -22235.39,E2 -22235.39} C_VEL
LIN {X 0,Y 186.545,Z 684.211,A -85,B 0,C 180,E1 -22238.671,E2 -22238.671} C_VEL
LIN {X 0,Y 186.304,Z 686.502,A -85,B 0,C 180,E1 -22241.249,E2 -22241.249} C_VEL
LIN {X 0,Y 186.441,Z 688.856,A -85,B 0,C 180,E1 -22245.303,E2 -22245.303} C_VEL
LIN {X 0,Y 186.785,Z 689.577,A -85,B 0,C 180,E1 -22247.522,E2 -22247.522} C_VEL
LIN {X 0,Y 187.622,Z 689.882,A -85,B 0,C 180,E1 -22250.537,E2 -22250.537} C_VEL
LIN {X 0,Y 189.101,Z 689.247,A -85,B 0,C 180,E1 -22254.134,E2 -22254.134} C_VEL
LIN {X 0,Y 190.278,Z 688.321,A -85,B 0,C 180,E1 -22256.313,E2 -22256.313} C_VEL
LIN {X 0,Y 191.69,Z 686.94,A -85,B 0,C 180,E1 -22258.469,E2 -22258.469} C_VEL
LIN {X 0,Y 194.153,Z 684.02,A -85,B 0,C 180,E1 -22261.663,E2 -22261.663} C_VEL
LIN {X 0,Y 197.32,Z 679.651,A -85,B 0,C 180,E1 -22264.997,E2 -22264.997} C_VEL
LIN {X 0,Y 201.114,Z 673.663,A -85,B 0,C 180,E1 -22268.341,E2 -22268.341} C_VEL
LIN {X 0,Y 204.937,Z 666.773,A -85,B 0,C 180,E1 -22271.249,E2 -22271.249} C_VEL
LIN {X 0,Y 208.584,Z 659.338,A -85,B 0,C 180,E1 -22273.691,E2 -22273.691} C_VEL
LIN {X 0,Y 212.735,Z 649.406,A -85,B 0,C 180,E1 -22276.268,E2 -22276.268} C_VEL
LIN {X 0,Y 214.131,Z 645.674,A -85,B 0,C 180,E1 -22277.075,E2 -22277.075} C_VEL
LIN {X 0,Y 214.376,Z 643.714,A -85,B 0,C 180,E1 -22277.602,E2 -22277.602} C_VEL
LIN {X 0,Y 210.389,Z 645.769,A -85,B 0,C 180,E1 -22278.081,E2 -22278.081} C_VEL
LIN {X 0,Y 204.258,Z 647.929,A -85,B 0,C 180,E1 -22279.177,E2 -22279.177} C_VEL
LIN {X 0,Y 198.461,Z 649.707,A -85,B 0,C 180,E1 -22280.401,E2 -22280.401} C_VEL
LIN {X 0,Y 193.1,Z 650.957,A -85,B 0,C 180,E1 -22281.778,E2 -22281.778} C_VEL
LIN {X 0,Y 192.328,Z 651.046,A -85,B 0,C 180,E1 -22282.261,E2 -22282.261} C_VEL
LIN {X 0,Y 191.982,Z 652.313,A -85,B 0,C 180,E1 -22282.678,E2 -22282.678} C_VEL
LIN {X 0,Y 190.46,Z 669.539,A -85,B 0,C 180,E1 -22284.63,E2 -22284.63} C_VEL
LIN {X 0,Y 189.135,Z 681.768,A -85,B 0,C 180,E1 -22286.446,E2 -22286.446} C_VEL
LIN {X 0,Y 187.606,Z 694.143,A -85,B 0,C 180,E1 -22288.811,E2 -22288.811} C_VEL
LIN {X 0,Y 186.346,Z 704.403,A -85,B 0,C 180,E1 -22291.259,E2 -22291.259} C_VEL
LIN {X 0,Y 185.203,Z 714.089,A -85,B 0,C 180,E1 -22294.127,E2 -22294.127} C_VEL
LIN {X 0,Y 184.401,Z 721.539,A -85,B 0,C 180,E1 -22296.797,E2 -22296.797} C_VEL
LIN {X 0,Y 183.742,Z 728.612,A -85,B 0,C 180,E1 -22299.865,E2 -22299.865} C_VEL
LIN {X 0,Y 183.282,Z 735.269,A -85,B 0,C 180,E1 -22303.474,E2 -22303.474} C_VEL
LIN {X 0,Y 183.166,Z 739.923,A -85,B 0,C 180,E1 -22306.691,E2 -22306.691} C_VEL
LIN {X 0,Y 183.391,Z 743.653,A -85,B 0,C 180,E1 -22310.07,E2 -22310.07} C_VEL
LIN {X 0,Y 184.146,Z 746.362,A -85,B 0,C 180,E1 -22313.426,E2 -22313.426} C_VEL
LIN {X 0,Y 185.77,Z 748.477,A -85,B 0,C 180,E1 -22317.833,E2 -22317.833} C_VEL
LIN {X 0,Y 186.985,Z 748.942,A -85,B 0,C 180,E1 -22320.001,E2 -22320.001} C_VEL
LIN {X 0,Y 190.188,Z 748.615,A -85,B 0,C 180,E1 -22324.239,E2 -22324.239} C_VEL
LIN {X 0,Y 194.401,Z 746.732,A -85,B 0,C 180,E1 -22328.315,E2 -22328.315} C_VEL
LIN {X 0,Y 198.217,Z 744.235,A -85,B 0,C 180,E1 -22331.246,E2 -22331.246} C_VEL
LIN {X 0,Y 203.105,Z 740.307,A -85,B 0,C 180,E1 -22334.32,E2 -22334.32} C_VEL
LIN {X 0,Y 209.233,Z 734.374,A -85,B 0,C 180,E1 -22337.597,E2 -22337.597} C_VEL
LIN {X 0,Y 214.801,Z 728.173,A -85,B 0,C 180,E1 -22340.094,E2 -22340.094} C_VEL
LIN {X 0,Y 221.498,Z 719.529,A -85,B 0,C 180,E1 -22342.739,E2 -22342.739} C_VEL
LIN {X 0,Y 227.146,Z 711.193,A -85,B 0,C 180,E1 -22344.69,E2 -22344.69} C_VEL
LIN {X 0,Y 233.31,Z 700.562,A -85,B 0,C 180,E1 -22346.621,E2 -22346.621} C_VEL
LIN {X 0,Y 238.653,Z 689.928,A -85,B 0,C 180,E1 -22348.111,E2 -22348.111} C_VEL
LIN {X 0,Y 243.5,Z 678.247,A -85,B 0,C 180,E1 -22349.385,E2 -22349.385} C_VEL
LIN {X 0,Y 248.04,Z 664.558,A -85,B 0,C 180,E1 -22350.514,E2 -22350.514} C_VEL
LIN {X 0,Y 251.302,Z 651.696,A -85,B 0,C 180,E1 -22351.28,E2 -22351.28} C_VEL
LIN {X 0,Y 251.941,Z 648.021,A -85,B 0,C 180,E1 -22351.608,E2 -22351.608} C_VEL
LIN {X 0,Y 252.995,Z 636.996,A -85,B 0,C 180,E1 -22353.366,E2 -22353.366} C_VEL
LIN {X 0,Y 253.632,Z 633.287,A -85,B 0,C 180,E1 -22353.653,E2 -22353.653} C_VEL
LIN {X 0,Y 258.8,Z 608.423,A -85,B 0,C 180,E1 -22354.665,E2 -22354.665} C_VEL
LIN {X 0,Y 258.493,Z 606.436,A -85,B 0,C 180,E1 -22356.738,E2 -22356.738} C_VEL
LIN {X 0,Y 258.507,Z 605.872,A -85,B 0,C 180,E1 -22358.705,E2 -22358.705} C_VEL
LIN {X 0,Y 258.901,Z 606.117,A -85,B 0,C 180,E1 -22360.628,E2 -22360.628} C_VEL
LIN {X 0,Y 256.874,Z 617.503,A -85,B 0,C 180,E1 -22361.74,E2 -22361.74} C_VEL
LIN {X 0,Y 255.328,Z 625.628,A -85,B 0,C 180,E1 -22362.306,E2 -22362.306} C_VEL
LIN {X 0,Y 247.711,Z 661.798,A -85,B 0,C 180,E1 -22363.801,E2 -22363.801} C_VEL
LIN {X 0,Y 243.476,Z 675.905,A -85,B 0,C 180,E1 -22364.549,E2 -22364.549} C_VEL
LIN {X 0,Y 238.91,Z 687.668,A -85,B 0,C 180,E1 -22365.364,E2 -22365.364} C_VEL
LIN {X 0,Y 233.38,Z 699.659,A -85,B 0,C 180,E1 -22366.508,E2 -22366.508} C_VEL
LIN {X 0,Y 227.697,Z 710.141,A -85,B 0,C 180,E1 -22367.767,E2 -22367.767} C_VEL
LIN {X 0,Y 221.346,Z 720.317,A -85,B 0,C 180,E1 -22369.387,E2 -22369.387} C_VEL
LIN {X 0,Y 214.404,Z 730.232,A -85,B 0,C 180,E1 -22371.475,E2 -22371.475} C_VEL
LIN {X 0,Y 207.886,Z 738.411,A -85,B 0,C 180,E1 -22373.724,E2 -22373.724} C_VEL
LIN {X 0,Y 200.89,Z 746.218,A -85,B 0,C 180,E1 -22376.56,E2 -22376.56} C_VEL
LIN {X 0,Y 194.676,Z 752.48,A -85,B 0,C 180,E1 -22379.637,E2 -22379.637} C_VEL
LIN {X 0,Y 188.588,Z 757.864,A -85,B 0,C 180,E1 -22383.432,E2 -22383.432} C_VEL
LIN {X 0,Y 183.862,Z 761.692,A -85,B 0,C 180,E1 -22387.524,E2 -22387.524} C_VEL
LIN {X 0,Y 180.17,Z 763.979,A -85,B 0,C 180,E1 -22391.813,E2 -22391.813} C_VEL
LIN {X 0,Y 177.785,Z 764.828,A -85,B 0,C 180,E1 -22396.276,E2 -22396.276} C_VEL
LIN {X 0,Y 176.648,Z 764.228,A -85,B 0,C 180,E1 -22400.839,E2 -22400.839} C_VEL
LIN {X 0,Y 176.649,Z 762.056,A -85,B 0,C 180,E1 -22405.432,E2 -22405.432} C_VEL
LIN {X 0,Y 177.128,Z 759.365,A -85,B 0,C 180,E1 -22408.859,E2 -22408.859} C_VEL
LIN {X 0,Y 177.273,Z 756.89,A -85,B 0,C 180,E1 -22411.132,E2 -22411.132} C_VEL
LIN {X 0,Y 177.209,Z 752.04,A -85,B 0,C 180,E1 -22414.546,E2 -22414.546} C_VEL
LIN {X 0,Y 177.298,Z 745.751,A -85,B 0,C 180,E1 -22417.97,E2 -22417.97} C_VEL
LIN {X 0,Y 177.639,Z 737.692,A -85,B 0,C 180,E1 -22421.405,E2 -22421.405} C_VEL
LIN {X 0,Y 178.368,Z 729.466,A -85,B 0,C 180,E1 -22424.252,E2 -22424.252} C_VEL
LIN {X 0,Y 179.442,Z 719.421,A -85,B 0,C 180,E1 -22427.078,E2 -22427.078} C_VEL
LIN {X 0,Y 180,Z 715.095,A -85,B 0,C 180,E1 -22428.197,E2 -22428.197} C_VEL
LIN {X 0,Y 181.496,Z 706.977,A -85,B 0,C 180,E1 -22431.213,E2 -22431.213} C_VEL
LIN {X 0,Y 183.447,Z 697.568,A -85,B 0,C 180,E1 -22434.016,E2 -22434.016} C_VEL
LIN {X 0,Y 185.696,Z 687.491,A -85,B 0,C 180,E1 -22436.4,E2 -22436.4} C_VEL
LIN {X 0,Y 187.871,Z 677.953,A -85,B 0,C 180,E1 -22438.178,E2 -22438.178} C_VEL
LIN {X 0,Y 189.815,Z 667.884,A -85,B 0,C 180,E1 -22439.68,E2 -22439.68} C_VEL
LIN {X 0,Y 191.694,Z 656.016,A -85,B 0,C 180,E1 -22441.031,E2 -22441.031} C_VEL
LIN {X 0,Y 193.1,Z 643.18,A -85,B 0,C 180,E1 -22442.079,E2 -22442.079} C_VEL
LIN {X 0,Y 193.963,Z 629.957,A -85,B 0,C 180,E1 -22442.764,E2 -22442.764} C_VEL
LIN {X 0,Y 194.608,Z 610.338,A -85,B 0,C 180,E1 -22443.476,E2 -22443.476} C_VEL
LIN {X 0,Y 190.988,Z 551.993,A -85,B 0,C 180,E1 -22446.503,E2 -22446.503} C_VEL
LIN {X 0,Y 189.813,Z 539.582,A -85,B 0,C 180,E1 -22447.244,E2 -22447.244} C_VEL
LIN {X 0,Y 183.77,Z 523.957,A -85,B 0,C 180,E1 -22449.102,E2 -22449.102} C_VEL
LIN {X 0,Y 182.606,Z 518.65,A -85,B 0,C 180,E1 -22451.285,E2 -22451.285} C_VEL
LIN {X 0,Y 180.061,Z 508.246,A -85,B 0,C 180,E1 -22456.146,E2 -22456.146} C_VEL
LIN {X 0,Y 178.445,Z 502.355,A -85,B 0,C 180,E1 -22459.213,E2 -22459.213} C_VEL
LIN {X 0,Y 178.414,Z 502.25,A -85,B 0,C 180,E1 -22463.78,E2 -22463.78} C_VEL
LIN {X 0,Y 178.476,Z 502.24,A -85,B 0,C 180,E1 -22466.544,E2 -22466.544} C_VEL
LIN {X 0,Y 178.512,Z 502.236,A -85,B 0,C 180,E1 -22470.004,E2 -22470.004} C_VEL
LIN {X 0,Y 178.524,Z 502.241,A -85,B 0,C 180,E1 -22474.873,E2 -22474.873} C_VEL
LIN {X 0,Y 178.612,Z 502.214,A -85,B 0,C 180,E1 -22480.782,E2 -22480.782} C_VEL
LIN {X 0,Y 178.654,Z 502.23,A -85,B 0,C 180,E1 -22484.015,E2 -22484.015} C_VEL
LIN {X 0,Y 178.85,Z 502.178,A -85,B 0,C 180,E1 -22489.208,E2 -22489.208} C_VEL
LIN {X 0,Y 178.916,Z 502.197,A -85,B 0,C 180,E1 -22493.232,E2 -22493.232} C_VEL
LIN {X 0,Y 179.141,Z 502.141,A -85,B 0,C 180,E1 -22497.751,E2 -22497.751} C_VEL
LIN {X 0,Y 179.357,Z 502.116,A -85,B 0,C 180,E1 -22499.999,E2 -22499.999} C_VEL
LIN {X 0,Y 178.861,Z 502.203,A -85,B 0,C 180,E1 -22504.506,E2 -22504.506} C_VEL
LIN {X 0,Y 178.925,Z 502.164,A -85,B 0,C 180,E1 -22509.039,E2 -22509.039} C_VEL
LIN {X 0,Y 178.675,Z 502.228,A -85,B 0,C 180,E1 -22513.65,E2 -22513.65} C_VEL
LIN {X 0,Y 178.637,Z 502.204,A -85,B 0,C 180,E1 -22518.344,E2 -22518.344} C_VEL
LIN {X 0,Y 178.499,Z 502.248,A -85,B 0,C 180,E1 -22523.186,E2 -22523.186} C_VEL
LIN {X 0,Y 178.475,Z 502.227,A -85,B 0,C 180,E1 -22528.198,E2 -22528.198} C_VEL
LIN {X 0,Y 178.468,Z 502.239,A -85,B 0,C 180,E1 -22530.792,E2 -22530.792} C_VEL
LIN {X 0,Y 178.473,Z 502.253,A -85,B 0,C 180,E1 -22534.221,E2 -22534.221} C_VEL
LIN {X 0,Y 178.389,Z 502.25,A -85,B 0,C 180,E1 -22539.075,E2 -22539.075} C_VEL
LIN {X 0,Y 178.409,Z 502.261,A -85,B 0,C 180,E1 -22542.041,E2 -22542.041} C_VEL
LIN {X 0,Y 178.451,Z 502.239,A -85,B 0,C 180,E1 -22545.144,E2 -22545.144} C_VEL
LIN {X 0,Y 178.496,Z 502.252,A -85,B 0,C 180,E1 -22548.424,E2 -22548.424} C_VEL
LIN {X 0,Y 178.459,Z 502.2,A -85,B 0,C 180,E1 -22553.797,E2 -22553.797} C_VEL
LIN {X 0,Y 178.483,Z 502.227,A -85,B 0,C 180,E1 -22556.551,E2 -22556.551} C_VEL
LIN {X 0,Y 178.515,Z 502.228,A -85,B 0,C 180,E1 -22560.009,E2 -22560.009} C_VEL
LIN {X 0,Y 178.537,Z 502.396,A -85,B 0,C 180,E1 -22564.872,E2 -22564.872} C_VEL
LIN {X 0,Y 178.807,Z 503.42,A -85,B 0,C 180,E1 -22565.305,E2 -22565.305} C_VEL
LIN {X 0,Y 180.237,Z 506.017,A -85,B 0,C 180,E1 -22565.761,E2 -22565.761} C_VEL
LIN {X 0,Y 187.507,Z 519.129,A -85,B 0,C 180,E1 -22567.815,E2 -22567.815} C_VEL
LIN {X 0,Y 193.201,Z 530.845,A -85,B 0,C 180,E1 -22569.354,E2 -22569.354} C_VEL
LIN {X 0,Y 197.016,Z 540.305,A -85,B 0,C 180,E1 -22570.39,E2 -22570.39} C_VEL
LIN {X 0,Y 195.778,Z 581.696,A -85,B 0,C 180,E1 -22571.908,E2 -22571.908} C_VEL
LIN {X 0,Y 195.27,Z 594.699,A -85,B 0,C 180,E1 -22572.632,E2 -22572.632} C_VEL
LIN {X 0,Y 194.372,Z 607.326,A -85,B 0,C 180,E1 -22573.73,E2 -22573.73} C_VEL
LIN {X 0,Y 192.914,Z 619.774,A -85,B 0,C 180,E1 -22575.229,E2 -22575.229} C_VEL
LIN {X 0,Y 190.946,Z 632.304,A -85,B 0,C 180,E1 -22577.246,E2 -22577.246} C_VEL
LIN {X 0,Y 188.823,Z 643.363,A -85,B 0,C 180,E1 -22579.55,E2 -22579.55} C_VEL
LIN {X 0,Y 186.944,Z 652.306,A -85,B 0,C 180,E1 -22581.899,E2 -22581.899} C_VEL
LIN {X 0,Y 184.696,Z 662.025,A -85,B 0,C 180,E1 -22585.092,E2 -22585.092} C_VEL
LIN {X 0,Y 183.165,Z 668.615,A -85,B 0,C 180,E1 -22587.805,E2 -22587.805} C_VEL
LIN {X 0,Y 181.554,Z 675.157,A -85,B 0,C 180,E1 -22591.113,E2 -22591.113} C_VEL
LIN {X 0,Y 180.383,Z 680.361,A -85,B 0,C 180,E1 -22594.473,E2 -22594.473} C_VEL
LIN {X 0,Y 179.615,Z 684.427,A -85,B 0,C 180,E1 -22597.875,E2 -22597.875} C_VEL
LIN {X 0,Y 179.249,Z 687.542,A -85,B 0,C 180,E1 -22601.425,E2 -22601.425} C_VEL
LIN {X 0,Y 179.476,Z 689.984,A -85,B 0,C 180,E1 -22605.913,E2 -22605.913} C_VEL
LIN {X 0,Y 179.895,Z 690.658,A -85,B 0,C 180,E1 -22608.216,E2 -22608.216} C_VEL
LIN {X 0,Y 180.747,Z 690.874,A -85,B 0,C 180,E1 -22611.064,E2 -22611.064} C_VEL
LIN {X 0,Y 182.5,Z 690.135,A -85,B 0,C 180,E1 -22615.066,E2 -22615.066} C_VEL
LIN {X 0,Y 184.971,Z 688.038,A -85,B 0,C 180,E1 -22619.088,E2 -22619.088} C_VEL
LIN {X 0,Y 187.98,Z 684.658,A -85,B 0,C 180,E1 -22622.831,E2 -22622.831} C_VEL
LIN {X 0,Y 191.137,Z 680.5,A -85,B 0,C 180,E1 -22626.041,E2 -22626.041} C_VEL
LIN {X 0,Y 194.774,Z 675.071,A -85,B 0,C 180,E1 -22629.161,E2 -22629.161} C_VEL
LIN {X 0,Y 198.825,Z 668.176,A -85,B 0,C 180,E1 -22632.195,E2 -22632.195} C_VEL
LIN {X 0,Y 202.555,Z 661.008,A -85,B 0,C 180,E1 -22634.641,E2 -22634.641} C_VEL
LIN {X 0,Y 206.696,Z 651.685,A -85,B 0,C 180,E1 -22637.155,E2 -22637.155} C_VEL
LIN {X 0,Y 200.589,Z 653.618,A -85,B 0,C 180,E1 -22638.265,E2 -22638.265} C_VEL
LIN {X 0,Y 192.399,Z 655.759,A -85,B 0,C 180,E1 -22640.098,E2 -22640.098} C_VEL
LIN {X 0,Y 189.472,Z 656.288,A -85,B 0,C 180,E1 -22640.909,E2 -22640.909} C_VEL
LIN {X 0,Y 186.668,Z 657.073,A -85,B 0,C 180,E1 -22641.596,E2 -22641.596} C_VEL
LIN {X 0,Y 184.976,Z 656.859,A -85,B 0,C 180,E1 -22642.391,E2 -22642.391} C_VEL
LIN {X 0,Y 184.54,Z 657.741,A -85,B 0,C 180,E1 -22642.879,E2 -22642.879} C_VEL
LIN {X 0,Y 184.198,Z 661.078,A -85,B 0,C 180,E1 -22643.346,E2 -22643.346} C_VEL
LIN {X 0,Y 182.869,Z 674.601,A -85,B 0,C 180,E1 -22645.134,E2 -22645.134} C_VEL
LIN {X 0,Y 181.44,Z 686.504,A -85,B 0,C 180,E1 -22647.162,E2 -22647.162} C_VEL
LIN {X 0,Y 180.114,Z 697.483,A -85,B 0,C 180,E1 -22649.52,E2 -22649.52} C_VEL
LIN {X 0,Y 178.74,Z 708.614,A -85,B 0,C 180,E1 -22652.484,E2 -22652.484} C_VEL
LIN {X 0,Y 177.675,Z 717.652,A -85,B 0,C 180,E1 -22655.482,E2 -22655.482} C_VEL
LIN {X 0,Y 176.825,Z 726.352,A -85,B 0,C 180,E1 -22659.041,E2 -22659.041} C_VEL
LIN {X 0,Y 176.309,Z 733.161,A -85,B 0,C 180,E1 -22662.563,E2 -22662.563} C_VEL
LIN {X 0,Y 176.111,Z 738.617,A -85,B 0,C 180,E1 -22666.147,E2 -22666.147} C_VEL
LIN {X 0,Y 176.237,Z 742.781,A -85,B 0,C 180,E1 -22669.663,E2 -22669.663} C_VEL
LIN {X 0,Y 176.97,Z 745.897,A -85,B 0,C 180,E1 -22673.158,E2 -22673.158} C_VEL
LIN {X 0,Y 178.575,Z 748.528,A -85,B 0,C 180,E1 -22677.745,E2 -22677.745} C_VEL
LIN {X 0,Y 181.258,Z 749.512,A -85,B 0,C 180,E1 -22682.223,E2 -22682.223} C_VEL
LIN {X 0,Y 185.049,Z 748.955,A -85,B 0,C 180,E1 -22686.543,E2 -22686.543} C_VEL
LIN {X 0,Y 187.334,Z 748.071,A -85,B 0,C 180,E1 -22688.631,E2 -22688.631} C_VEL
LIN {X 0,Y 189.892,Z 746.768,A -85,B 0,C 180,E1 -22690.665,E2 -22690.665} C_VEL
LIN {X 0,Y 195.816,Z 742.951,A -85,B 0,C 180,E1 -22694.551,E2 -22694.551} C_VEL
LIN {X 0,Y 200.829,Z 738.908,A -85,B 0,C 180,E1 -22697.306,E2 -22697.306} C_VEL
LIN {X 0,Y 206.373,Z 733.69,A -85,B 0,C 180,E1 -22699.911,E2 -22699.911} C_VEL
LIN {X 0,Y 213.377,Z 726.129,A -85,B 0,C 180,E1 -22702.738,E2 -22702.738} C_VEL
LIN {X 0,Y 218.805,Z 719.332,A -85,B 0,C 180,E1 -22704.681,E2 -22704.681} C_VEL
LIN {X 0,Y 225.666,Z 709.6,A -85,B 0,C 180,E1 -22706.846,E2 -22706.846} C_VEL
LIN {X 0,Y 231.788,Z 699.394,A -85,B 0,C 180,E1 -22708.576,E2 -22708.576} C_VEL
LIN {X 0,Y 237.93,Z 687.214,A -85,B 0,C 180,E1 -22710.143,E2 -22710.143} C_VEL
LIN {X 0,Y 243.024,Z 674.946,A -85,B 0,C 180,E1 -22711.369,E2 -22711.369} C_VEL
LIN {X 0,Y 247.261,Z 661.903,A -85,B 0,C 180,E1 -22712.325,E2 -22712.325} C_VEL
LIN {X 0,Y 250.413,Z 648.943,A -85,B 0,C 180,E1 -22713.013,E2 -22713.013} C_VEL
LIN {X 0,Y 253.632,Z 633.287,A -85,B 0,C 180,E1 -22713.653,E2 -22713.653} C_VEL
LIN {X 0,Y 254.313,Z 629.581,A -85,B 0,C 180,E1 -22713.951,E2 -22713.951} C_VEL
LIN {X 0,Y 255.951,Z 618.649,A -85,B 0,C 180,E1 -22715.713,E2 -22715.713} C_VEL
LIN {X 0,Y 256.706,Z 614.941,A -85,B 0,C 180,E1 -22715.984,E2 -22715.984} C_VEL
LIN {X 0,Y 256.919,Z 613.954,A -85,B 0,C 180,E1 -22716.045,E2 -22716.045} C_VEL
LIN {X 0,Y 256.868,Z 613,A -85,B 0,C 180,E1 -22717.487,E2 -22717.487} C_VEL
LIN {X 0,Y 257.078,Z 612.85,A -85,B 0,C 180,E1 -22719.605,E2 -22719.605} C_VEL
LIN {X 0,Y 255.231,Z 621.727,A -85,B 0,C 180,E1 -22720.418,E2 -22720.418} C_VEL
LIN {X 0,Y 253.982,Z 627.753,A -85,B 0,C 180,E1 -22720.789,E2 -22720.789} C_VEL
LIN {X 0,Y 246.957,Z 660.033,A -85,B 0,C 180,E1 -22722.091,E2 -22722.091} C_VEL
LIN {X 0,Y 242.511,Z 674.406,A -85,B 0,C 180,E1 -22722.811,E2 -22722.811} C_VEL
LIN {X 0,Y 236.983,Z 688.052,A -85,B 0,C 180,E1 -22723.705,E2 -22723.705} C_VEL
LIN {X 0,Y 231.403,Z 699.584,A -85,B 0,C 180,E1 -22724.767,E2 -22724.767} C_VEL
LIN {X 0,Y 223.917,Z 712.336,A -85,B 0,C 180,E1 -22726.326,E2 -22726.326} C_VEL
LIN {X 0,Y 217.487,Z 721.872,A -85,B 0,C 180,E1 -22727.889,E2 -22727.889} C_VEL
LIN {X 0,Y 210.24,Z 731.308,A -85,B 0,C 180,E1 -22729.943,E2 -22729.943} C_VEL
LIN {X 0,Y 202.353,Z 740.354,A -85,B 0,C 180,E1 -22732.566,E2 -22732.566} C_VEL
LIN {X 0,Y 196.101,Z 746.697,A -85,B 0,C 180,E1 -22735.007,E2 -22735.007} C_VEL
LIN {X 0,Y 188.65,Z 753.381,A -85,B 0,C 180,E1 -22738.559,E2 -22738.559} C_VEL
LIN {X 0,Y 183.841,Z 757.262,A -85,B 0,C 180,E1 -22741.45,E2 -22741.45} C_VEL
LIN {X 0,Y 179.652,Z 760.243,A -85,B 0,C 180,E1 -22744.508,E2 -22744.508} C_VEL
LIN {X 0,Y 175.234,Z 762.942,A -85,B 0,C 180,E1 -22748.837,E2 -22748.837} C_VEL
LIN {X 0,Y 171.915,Z 764.204,A -85,B 0,C 180,E1 -22753.368,E2 -22753.368} C_VEL
LIN {X 0,Y 170.111,Z 763.992,A -85,B 0,C 180,E1 -22758.075,E2 -22758.075} C_VEL
LIN {X 0,Y 169.548,Z 762.359,A -85,B 0,C 180,E1 -22762.853,E2 -22762.853} C_VEL
LIN {X 0,Y 169.649,Z 760.954,A -85,B 0,C 180,E1 -22765.243,E2 -22765.243} C_VEL
LIN {X 0,Y 170.169,Z 758.015,A -85,B 0,C 180,E1 -22768.813,E2 -22768.813} C_VEL
LIN {X 0,Y 170.302,Z 755.388,A -85,B 0,C 180,E1 -22771.178,E2 -22771.178} C_VEL
LIN {X 0,Y 170.239,Z 750.286,A -85,B 0,C 180,E1 -22774.732,E2 -22774.732} C_VEL
LIN {X 0,Y 170.319,Z 744.323,A -85,B 0,C 180,E1 -22777.97,E2 -22777.97} C_VEL
LIN {X 0,Y 170.64,Z 736.735,A -85,B 0,C 180,E1 -22781.278,E2 -22781.278} C_VEL
LIN {X 0,Y 171.369,Z 728.412,A -85,B 0,C 180,E1 -22784.241,E2 -22784.241} C_VEL
LIN {X 0,Y 172.585,Z 717.126,A -85,B 0,C 180,E1 -22787.473,E2 -22787.473} C_VEL
LIN {X 0,Y 174.349,Z 707.631,A -85,B 0,C 180,E1 -22791.267,E2 -22791.267} C_VEL
LIN {X 0,Y 176.466,Z 697.788,A -85,B 0,C 180,E1 -22794.401,E2 -22794.401} C_VEL
LIN {X 0,Y 179.028,Z 686.749,A -85,B 0,C 180,E1 -22797.148,E2 -22797.148} C_VEL
LIN {X 0,Y 181.262,Z 677.256,A -85,B 0,C 180,E1 -22798.985,E2 -22798.985} C_VEL
LIN {X 0,Y 183.62,Z 665.336,A -85,B 0,C 180,E1 -22800.787,E2 -22800.787} C_VEL
LIN {X 0,Y 185.552,Z 653.026,A -85,B 0,C 180,E1 -22802.165,E2 -22802.165} C_VEL
LIN {X 0,Y 187.023,Z 639.895,A -85,B 0,C 180,E1 -22803.197,E2 -22803.197} C_VEL
LIN {X 0,Y 187.769,Z 625.695,A -85,B 0,C 180,E1 -22803.876,E2 -22803.876} C_VEL
LIN {X 0,Y 188.264,Z 610.673,A -85,B 0,C 180,E1 -22804.439,E2 -22804.439} C_VEL
LIN {X 0,Y 184.772,Z 552.36,A -85,B 0,C 180,E1 -22807.589,E2 -22807.589} C_VEL
LIN {X 0,Y 183.816,Z 541.792,A -85,B 0,C 180,E1 -22808.244,E2 -22808.244} C_VEL
LIN {X 0,Y 177.847,Z 526.574,A -85,B 0,C 180,E1 -22810.133,E2 -22810.133} C_VEL
LIN {X 0,Y 176.225,Z 522.376,A -85,B 0,C 180,E1 -22810.787,E2 -22810.787} C_VEL
LIN {X 0,Y 174.108,Z 513.267,A -85,B 0,C 180,E1 -22815.056,E2 -22815.056} C_VEL
LIN {X 0,Y 171.395,Z 503.28,A -85,B 0,C 180,E1 -22820.357,E2 -22820.357} C_VEL
LIN {X 0,Y 171.389,Z 503.117,A -85,B 0,C 180,E1 -22825.089,E2 -22825.089} C_VEL
LIN {X 0,Y 171.438,Z 503.109,A -85,B 0,C 180,E1 -22830.531,E2 -22830.531} C_VEL
LIN {X 0,Y 171.448,Z 503.128,A -85,B 0,C 180,E1 -22835.799,E2 -22835.799} C_VEL
LIN {X 0,Y 171.568,Z 503.091,A -85,B 0,C 180,E1 -22840.869,E2 -22840.869} C_VEL
LIN {X 0,Y 171.598,Z 503.105,A -85,B 0,C 180,E1 -22845.774,E2 -22845.774} C_VEL
LIN {X 0,Y 171.88,Z 503.053,A -85,B 0,C 180,E1 -22850.586,E2 -22850.586} C_VEL
LIN {X 0,Y 171.81,Z 503.078,A -85,B 0,C 180,E1 -22855.306,E2 -22855.306} C_VEL
LIN {X 0,Y 172.32,Z 502.991,A -85,B 0,C 180,E1 -22859.999,E2 -22859.999} C_VEL
LIN {X 0,Y 171.81,Z 503.08,A -85,B 0,C 180,E1 -22864.692,E2 -22864.692} C_VEL
LIN {X 0,Y 171.861,Z 503.043,A -85,B 0,C 180,E1 -22869.414,E2 -22869.414} C_VEL
LIN {X 0,Y 171.597,Z 503.11,A -85,B 0,C 180,E1 -22874.225,E2 -22874.225} C_VEL
LIN {X 0,Y 171.532,Z 503.085,A -85,B 0,C 180,E1 -22879.562,E2 -22879.562} C_VEL
LIN {X 0,Y 171.457,Z 503.123,A -85,B 0,C 180,E1 -22885.618,E2 -22885.618} C_VEL
LIN {X 0,Y 171.43,Z 503.112,A -85,B 0,C 180,E1 -22890.588,E2 -22890.588} C_VEL
LIN {X 0,Y 171.381,Z 503.129,A -85,B 0,C 180,E1 -22895.036,E2 -22895.036} C_VEL
LIN {X 0,Y 171.35,Z 503.124,A -85,B 0,C 180,E1 -22898.811,E2 -22898.811} C_VEL
LIN {X 0,Y 171.357,Z 503.122,A -85,B 0,C 180,E1 -22904.204,E2 -22904.204} C_VEL
LIN {X 0,Y 171.415,Z 503.129,A -85,B 0,C 180,E1 -22909.01,E2 -22909.01} C_VEL
LIN {X 0,Y 171.431,Z 503.08,A -85,B 0,C 180,E1 -22912.058,E2 -22912.058} C_VEL
LIN {X 0,Y 171.42,Z 503.13,A -85,B 0,C 180,E1 -22917.798,E2 -22917.798} C_VEL
LIN {X 0,Y 171.418,Z 503.142,A -85,B 0,C 180,E1 -22922.868,E2 -22922.868} C_VEL
LIN {X 0,Y 171.526,Z 503.71,A -85,B 0,C 180,E1 -22923.557,E2 -22923.557} C_VEL
LIN {X 0,Y 172.878,Z 506.59,A -85,B 0,C 180,E1 -22924.159,E2 -22924.159} C_VEL
LIN {X 0,Y 173.995,Z 508.232,A -85,B 0,C 180,E1 -22924.5,E2 -22924.5} C_VEL
LIN {X 0,Y 180.51,Z 519.768,A -85,B 0,C 180,E1 -22926.469,E2 -22926.469} C_VEL
LIN {X 0,Y 186.777,Z 532.312,A -85,B 0,C 180,E1 -22928.268,E2 -22928.268} C_VEL
LIN {X 0,Y 190.764,Z 542.026,A -85,B 0,C 180,E1 -22929.412,E2 -22929.412} C_VEL
LIN {X 0,Y 189.477,Z 584.724,A -85,B 0,C 180,E1 -22931.053,E2 -22931.053} C_VEL
LIN {X 0,Y 188.817,Z 597.983,A -85,B 0,C 180,E1 -22931.868,E2 -22931.868} C_VEL
LIN {X 0,Y 187.772,Z 609.984,A -85,B 0,C 180,E1 -22933.002,E2 -22933.002} C_VEL
LIN {X 0,Y 186.165,Z 622.815,A -85,B 0,C 180,E1 -22934.681,E2 -22934.681} C_VEL
LIN {X 0,Y 184.356,Z 633.545,A -85,B 0,C 180,E1 -22936.501,E2 -22936.501} C_VEL
LIN {X 0,Y 182.158,Z 644.532,A -85,B 0,C 180,E1 -22938.881,E2 -22938.881} C_VEL
LIN {X 0,Y 179.971,Z 654.334,A -85,B 0,C 180,E1 -22941.583,E2 -22941.583} C_VEL
LIN {X 0,Y 178.002,Z 662.401,A -85,B 0,C 180,E1 -22944.339,E2 -22944.339} C_VEL
LIN {X 0,Y 176.05,Z 670.332,A -85,B 0,C 180,E1 -22947.716,E2 -22947.716} C_VEL
LIN {X 0,Y 174.436,Z 676.696,A -85,B 0,C 180,E1 -22951.158,E2 -22951.158} C_VEL
LIN {X 0,Y 173.259,Z 681.78,A -85,B 0,C 180,E1 -22954.657,E2 -22954.657} C_VEL
LIN {X 0,Y 172.504,Z 685.745,A -85,B 0,C 180,E1 -22958.202,E2 -22958.202} C_VEL
LIN {X 0,Y 172.198,Z 688.684,A -85,B 0,C 180,E1 -22961.779,E2 -22961.779} C_VEL
LIN {X 0,Y 172.267,Z 690.093,A -85,B 0,C 180,E1 -22964.173,E2 -22964.173} C_VEL
LIN {X 0,Y 172.524,Z 691.113,A -85,B 0,C 180,E1 -22966.572,E2 -22966.572} C_VEL
LIN {X 0,Y 173.027,Z 691.713,A -85,B 0,C 180,E1 -22968.966,E2 -22968.966} C_VEL
LIN {X 0,Y 174.73,Z 691.65,A -85,B 0,C 180,E1 -22973.721,E2 -22973.721} C_VEL
LIN {X 0,Y 175.94,Z 691.025,A -85,B 0,C 180,E1 -22976.07,E2 -22976.07} C_VEL
LIN {X 0,Y 178.4,Z 689.007,A -85,B 0,C 180,E1 -22979.926,E2 -22979.926} C_VEL
LIN {X 0,Y 181.897,Z 685.295,A -85,B 0,C 180,E1 -22984.077,E2 -22984.077} C_VEL
LIN {X 0,Y 185.287,Z 681.024,A -85,B 0,C 180,E1 -22987.369,E2 -22987.369} C_VEL
LIN {X 0,Y 189.154,Z 675.475,A -85,B 0,C 180,E1 -22990.562,E2 -22990.562} C_VEL
LIN {X 0,Y 193.451,Z 668.381,A -85,B 0,C 180,E1 -22993.655,E2 -22993.655} C_VEL
LIN {X 0,Y 198.095,Z 659.642,A -85,B 0,C 180,E1 -22996.551,E2 -22996.551} C_VEL
LIN {X 0,Y 198.176,Z 658.618,A -85,B 0,C 180,E1 -22996.985,E2 -22996.985} C_VEL
LIN {X 0,Y 190.943,Z 660.457,A -85,B 0,C 180,E1 -22998.509,E2 -22998.509} C_VEL
LIN {X 0,Y 185.479,Z 661.588,A -85,B 0,C 180,E1 -22999.899,E2 -22999.899} C_VEL
LIN {X 0,Y 178.437,Z 662.618,A -85,B 0,C 180,E1 -23002.113,E2 -23002.113} C_VEL
LIN {X 0,Y 177.266,Z 662.449,A -85,B 0,C 180,E1 -23002.88,E2 -23002.88} C_VEL
LIN {X 0,Y 176.864,Z 663.804,A -85,B 0,C 180,E1 -23003.413,E2 -23003.413} C_VEL
LIN {X 0,Y 175.352,Z 678.094,A -85,B 0,C 180,E1 -23005.521,E2 -23005.521} C_VEL
LIN {X 0,Y 173.901,Z 689.886,A -85,B 0,C 180,E1 -23007.754,E2 -23007.754} C_VEL
LIN {X 0,Y 172.507,Z 701.087,A -85,B 0,C 180,E1 -23010.399,E2 -23010.399} C_VEL
LIN {X 0,Y 171.364,Z 710.613,A -85,B 0,C 180,E1 -23013.185,E2 -23013.185} C_VEL
LIN {X 0,Y 170.373,Z 719.287,A -85,B 0,C 180,E1 -23016.286,E2 -23016.286} C_VEL
LIN {X 0,Y 169.684,Z 726.416,A -85,B 0,C 180,E1 -23019.388,E2 -23019.388} C_VEL
LIN {X 0,Y 169.219,Z 733.366,A -85,B 0,C 180,E1 -23023.1,E2 -23023.1} C_VEL
LIN {X 0,Y 169.032,Z 738.81,A -85,B 0,C 180,E1 -23026.782,E2 -23026.782} C_VEL
LIN {X 0,Y 169.257,Z 743.037,A -85,B 0,C 180,E1 -23030.44,E2 -23030.44} C_VEL
LIN {X 0,Y 169.873,Z 745.534,A -85,B 0,C 180,E1 -23033.211,E2 -23033.211} C_VEL
LIN {X 0,Y 171.356,Z 748.389,A -85,B 0,C 180,E1 -23037.65,E2 -23037.65} C_VEL
LIN {X 0,Y 174.062,Z 749.895,A -85,B 0,C 180,E1 -23042.315,E2 -23042.315} C_VEL
LIN {X 0,Y 176.445,Z 750.048,A -85,B 0,C 180,E1 -23045.232,E2 -23045.232} C_VEL
LIN {X 0,Y 180.256,Z 749.232,A -85,B 0,C 180,E1 -23048.973,E2 -23048.973} C_VEL
LIN {X 0,Y 185.809,Z 746.833,A -85,B 0,C 180,E1 -23053.118,E2 -23053.118} C_VEL
LIN {X 0,Y 189.576,Z 744.617,A -85,B 0,C 180,E1 -23055.436,E2 -23055.436} C_VEL
LIN {X 0,Y 196.004,Z 740.015,A -85,B 0,C 180,E1 -23058.828,E2 -23058.828} C_VEL
LIN {X 0,Y 201.904,Z 735.021,A -85,B 0,C 180,E1 -23061.439,E2 -23061.439} C_VEL
LIN {X 0,Y 209.081,Z 727.84,A -85,B 0,C 180,E1 -23064.202,E2 -23064.202} C_VEL
LIN {X 0,Y 214.983,Z 721.137,A -85,B 0,C 180,E1 -23066.189,E2 -23066.189} C_VEL
LIN {X 0,Y 222.17,Z 711.675,A -85,B 0,C 180,E1 -23068.328,E2 -23068.328} C_VEL
LIN {X 0,Y 228.965,Z 701.199,A -85,B 0,C 180,E1 -23070.132,E2 -23070.132} C_VEL
LIN {X 0,Y 235,Z 690.231,A -85,B 0,C 180,E1 -23071.559,E2 -23071.559} C_VEL
LIN {X 0,Y 240.93,Z 676.862,A -85,B 0,C 180,E1 -23072.909,E2 -23072.909} C_VEL
LIN {X 0,Y 245.636,Z 663.539,A -85,B 0,C 180,E1 -23073.887,E2 -23073.887} C_VEL
LIN {X 0,Y 249,Z 650.909,A -85,B 0,C 180,E1 -23074.551,E2 -23074.551} C_VEL
LIN {X 0,Y 256.706,Z 614.941,A -85,B 0,C 180,E1 -23075.984,E2 -23075.984} C_VEL
LIN {X 0,Y 256.824,Z 614.275,A -85,B 0,C 180,E1 -23076.167,E2 -23076.167} C_VEL
LIN {X 0,Y 256.682,Z 614.542,A -85,B 0,C 180,E1 -23076.662,E2 -23076.662} C_VEL
LIN {X 0,Y 256.047,Z 616.906,A -85,B 0,C 180,E1 -23077.476,E2 -23077.476} C_VEL
LIN {X 0,Y 254.55,Z 623.267,A -85,B 0,C 180,E1 -23078.616,E2 -23078.616} C_VEL
LIN {X 0,Y 253.432,Z 628.254,A -85,B 0,C 180,E1 -23079.158,E2 -23079.158} C_VEL
LIN {X 0,Y 253.034,Z 630.038,A -85,B 0,C 180,E1 -23079.259,E2 -23079.259} C_VEL
LIN {X 0,Y 246.291,Z 659.29,A -85,B 0,C 180,E1 -23080.397,E2 -23080.397} C_VEL
LIN {X 0,Y 241.445,Z 674.399,A -85,B 0,C 180,E1 -23081.13,E2 -23081.13} C_VEL
LIN {X 0,Y 236.098,Z 687.129,A -85,B 0,C 180,E1 -23081.907,E2 -23081.907} C_VEL
LIN {X 0,Y 229.546,Z 699.869,A -85,B 0,C 180,E1 -23083.028,E2 -23083.028} C_VEL
LIN {X 0,Y 222.04,Z 712.078,A -85,B 0,C 180,E1 -23084.475,E2 -23084.475} C_VEL
LIN {X 0,Y 215.077,Z 721.788,A -85,B 0,C 180,E1 -23086.018,E2 -23086.018} C_VEL
LIN {X 0,Y 206.257,Z 732.474,A -85,B 0,C 180,E1 -23088.357,E2 -23088.357} C_VEL
LIN {X 0,Y 199.178,Z 739.997,A -85,B 0,C 180,E1 -23090.566,E2 -23090.566} C_VEL
LIN {X 0,Y 192.517,Z 746.223,A -85,B 0,C 180,E1 -23092.958,E2 -23092.958} C_VEL
LIN {X 0,Y 186.451,Z 751.404,A -85,B 0,C 180,E1 -23095.566,E2 -23095.566} C_VEL
LIN {X 0,Y 180.982,Z 755.545,A -85,B 0,C 180,E1 -23098.379,E2 -23098.379} C_VEL
LIN {X 0,Y 175.533,Z 759.141,A -85,B 0,C 180,E1 -23101.745,E2 -23101.745} C_VEL
LIN {X 0,Y 170.821,Z 761.834,A -85,B 0,C 180,E1 -23105.702,E2 -23105.702} C_VEL
LIN {X 0,Y 166.718,Z 763.43,A -85,B 0,C 180,E1 -23110.287,E2 -23110.287} C_VEL
LIN {X 0,Y 165.109,Z 763.703,A -85,B 0,C 180,E1 -23112.661,E2 -23112.661} C_VEL
LIN {X 0,Y 163.176,Z 763.231,A -85,B 0,C 180,E1 -23117.56,E2 -23117.56} C_VEL
LIN {X 0,Y 162.564,Z 761.269,A -85,B 0,C 180,E1 -23122.544,E2 -23122.544} C_VEL
LIN {X 0,Y 162.666,Z 759.718,A -85,B 0,C 180,E1 -23125.039,E2 -23125.039} C_VEL
LIN {X 0,Y 163.219,Z 756.574,A -85,B 0,C 180,E1 -23128.762,E2 -23128.762} C_VEL
LIN {X 0,Y 163.327,Z 753.759,A -85,B 0,C 180,E1 -23131.229,E2 -23131.229} C_VEL
LIN {X 0,Y 163.274,Z 748.358,A -85,B 0,C 180,E1 -23134.934,E2 -23134.934} C_VEL
LIN {X 0,Y 163.388,Z 741.99,A -85,B 0,C 180,E1 -23138.373,E2 -23138.373} C_VEL
LIN {X 0,Y 163.765,Z 734.169,A -85,B 0,C 180,E1 -23141.758,E2 -23141.758} C_VEL
LIN {X 0,Y 164.548,Z 725.395,A -85,B 0,C 180,E1 -23144.844,E2 -23144.844} C_VEL
LIN {X 0,Y 165.408,Z 717.256,A -85,B 0,C 180,E1 -23147.298,E2 -23147.298} C_VEL
LIN {X 0,Y 166.932,Z 709.082,A -85,B 0,C 180,E1 -23150.964,E2 -23150.964} C_VEL
LIN {X 0,Y 168.796,Z 700.852,A -85,B 0,C 180,E1 -23153.92,E2 -23153.92} C_VEL
LIN {X 0,Y 171.243,Z 690.679,A -85,B 0,C 180,E1 -23156.832,E2 -23156.832} C_VEL
LIN {X 0,Y 174.069,Z 679.43,A -85,B 0,C 180,E1 -23159.306,E2 -23159.306} C_VEL
LIN {X 0,Y 176.426,Z 668.367,A -85,B 0,C 180,E1 -23161.184,E2 -23161.184} C_VEL
LIN {X 0,Y 178.651,Z 656.168,A -85,B 0,C 180,E1 -23162.741,E2 -23162.741} C_VEL
LIN {X 0,Y 180.277,Z 643.265,A -85,B 0,C 180,E1 -23163.931,E2 -23163.931} C_VEL
LIN {X 0,Y 181.33,Z 629.5,A -85,B 0,C 180,E1 -23164.732,E2 -23164.732} C_VEL
LIN {X 0,Y 182.003,Z 611.447,A -85,B 0,C 180,E1 -23165.438,E2 -23165.438} C_VEL
LIN {X 0,Y 178.6,Z 551.527,A -85,B 0,C 180,E1 -23168.811,E2 -23168.811} C_VEL
LIN {X 0,Y 177.877,Z 543.943,A -85,B 0,C 180,E1 -23169.314,E2 -23169.314} C_VEL
LIN {X 0,Y 172.032,Z 529.075,A -85,B 0,C 180,E1 -23171.283,E2 -23171.283} C_VEL
LIN {X 0,Y 168.722,Z 521.168,A -85,B 0,C 180,E1 -23172.557,E2 -23172.557} C_VEL
LIN {X 0,Y 166.657,Z 512.655,A -85,B 0,C 180,E1 -23176.842,E2 -23176.842} C_VEL
LIN {X 0,Y 164.356,Z 504.156,A -85,B 0,C 180,E1 -23181.68,E2 -23181.68} C_VEL
LIN {X 0,Y 164.317,Z 504,A -85,B 0,C 180,E1 -23186.218,E2 -23186.218} C_VEL
LIN {X 0,Y 164.379,Z 504.005,A -85,B 0,C 180,E1 -23189.131,E2 -23189.131} C_VEL
LIN {X 0,Y 164.406,Z 503.997,A -85,B 0,C 180,E1 -23194.691,E2 -23194.691} C_VEL
LIN {X 0,Y 164.474,Z 503.972,A -85,B 0,C 180,E1 -23200.049,E2 -23200.049} C_VEL
LIN {X 0,Y 164.542,Z 503.987,A -85,B 0,C 180,E1 -23205.15,E2 -23205.15} C_VEL
LIN {X 0,Y 164.794,Z 503.931,A -85,B 0,C 180,E1 -23210.177,E2 -23210.177} C_VEL
LIN {X 0,Y 164.842,Z 503.948,A -85,B 0,C 180,E1 -23212.651,E2 -23212.651} C_VEL
LIN {X 0,Y 165.037,Z 503.896,A -85,B 0,C 180,E1 -23217.558,E2 -23217.558} C_VEL
LIN {X 0,Y 165.283,Z 503.866,A -85,B 0,C 180,E1 -23219.999,E2 -23219.999} C_VEL
LIN {X 0,Y 164.759,Z 503.957,A -85,B 0,C 180,E1 -23224.893,E2 -23224.893} C_VEL
LIN {X 0,Y 164.834,Z 503.924,A -85,B 0,C 180,E1 -23227.348,E2 -23227.348} C_VEL
LIN {X 0,Y 164.738,Z 503.943,A -85,B 0,C 180,E1 -23231.146,E2 -23231.146} C_VEL
LIN {X 0,Y 164.493,Z 503.972,A -85,B 0,C 180,E1 -23237.401,E2 -23237.401} C_VEL
LIN {X 0,Y 164.461,Z 503.966,A -85,B 0,C 180,E1 -23239.99,E2 -23239.99} C_VEL
LIN {X 0,Y 164.381,Z 503.998,A -85,B 0,C 180,E1 -23246.135,E2 -23246.135} C_VEL
LIN {X 0,Y 164.364,Z 503.998,A -85,B 0,C 180,E1 -23251.229,E2 -23251.229} C_VEL
LIN {X 0,Y 164.284,Z 503.997,A -85,B 0,C 180,E1 -23256.791,E2 -23256.791} C_VEL
LIN {X 0,Y 164.284,Z 504.014,A -85,B 0,C 180,E1 -23259.917,E2 -23259.917} C_VEL
LIN {X 0,Y 164.296,Z 504.006,A -85,B 0,C 180,E1 -23263.354,E2 -23263.354} C_VEL
LIN {X 0,Y 164.347,Z 504.008,A -85,B 0,C 180,E1 -23266.832,E2 -23266.832} C_VEL
LIN {X 0,Y 164.364,Z 503.983,A -85,B 0,C 180,E1 -23270.322,E2 -23270.322} C_VEL
LIN {X 0,Y 164.339,Z 503.956,A -85,B 0,C 180,E1 -23274.343,E2 -23274.343} C_VEL
LIN {X 0,Y 164.398,Z 503.997,A -85,B 0,C 180,E1 -23279.141,E2 -23279.141} C_VEL
LIN {X 0,Y 164.452,Z 504.255,A -85,B 0,C 180,E1 -23281.617,E2 -23281.617} C_VEL
LIN {X 0,Y 164.759,Z 505.439,A -85,B 0,C 180,E1 -23282.062,E2 -23282.062} C_VEL
LIN {X 0,Y 166.35,Z 508.069,A -85,B 0,C 180,E1 -23282.642,E2 -23282.642} C_VEL
LIN {X 0,Y 172.901,Z 519.212,A -85,B 0,C 180,E1 -23284.802,E2 -23284.802} C_VEL
LIN {X 0,Y 180.836,Z 534.736,A -85,B 0,C 180,E1 -23287.234,E2 -23287.234} C_VEL
LIN {X 0,Y 184.483,Z 543.282,A -85,B 0,C 180,E1 -23288.332,E2 -23288.332} C_VEL
LIN {X 0,Y 183.218,Z 588.818,A -85,B 0,C 180,E1 -23290.202,E2 -23290.202} C_VEL
LIN {X 0,Y 182.365,Z 601.608,A -85,B 0,C 180,E1 -23291.11,E2 -23291.11} C_VEL
LIN {X 0,Y 181.068,Z 614.656,A -85,B 0,C 180,E1 -23292.498,E2 -23292.498} C_VEL
LIN {X 0,Y 179.43,Z 625.838,A -85,B 0,C 180,E1 -23294.091,E2 -23294.091} C_VEL
LIN {X 0,Y 177.255,Z 637.416,A -85,B 0,C 180,E1 -23296.242,E2 -23296.242} C_VEL
LIN {X 0,Y 175.028,Z 647.828,A -85,B 0,C 180,E1 -23298.716,E2 -23298.716} C_VEL
LIN {X 0,Y 173.009,Z 656.362,A -85,B 0,C 180,E1 -23301.242,E2 -23301.242} C_VEL
LIN {X 0,Y 171.003,Z 664.252,A -85,B 0,C 180,E1 -23304.107,E2 -23304.107} C_VEL
LIN {X 0,Y 168.949,Z 671.992,A -85,B 0,C 180,E1 -23307.62,E2 -23307.62} C_VEL
LIN {X 0,Y 167.312,Z 678.224,A -85,B 0,C 180,E1 -23311.207,E2 -23311.207} C_VEL
LIN {X 0,Y 166.12,Z 683.201,A -85,B 0,C 180,E1 -23314.858,E2 -23314.858} C_VEL
LIN {X 0,Y 165.408,Z 687.061,A -85,B 0,C 180,E1 -23318.556,E2 -23318.556} C_VEL
LIN {X 0,Y 165.172,Z 689.9,A -85,B 0,C 180,E1 -23322.287,E2 -23322.287} C_VEL
LIN {X 0,Y 165.264,Z 691.269,A -85,B 0,C 180,E1 -23324.787,E2 -23324.787} C_VEL
LIN {X 0,Y 165.606,Z 692.232,A -85,B 0,C 180,E1 -23327.286,E2 -23327.286} C_VEL
LIN {X 0,Y 167.037,Z 692.862,A -85,B 0,C 180,E1 -23332.255,E2 -23332.255} C_VEL
LIN {X 0,Y 168.115,Z 692.588,A -85,B 0,C 180,E1 -23334.715,E2 -23334.715} C_VEL
LIN {X 0,Y 169.419,Z 691.884,A -85,B 0,C 180,E1 -23337.154,E2 -23337.154} C_VEL
LIN {X 0,Y 171.902,Z 689.959,A -85,B 0,C 180,E1 -23340.847,E2 -23340.847} C_VEL
LIN {X 0,Y 174.792,Z 687.148,A -85,B 0,C 180,E1 -23344.261,E2 -23344.261} C_VEL
LIN {X 0,Y 178.855,Z 682.399,A -85,B 0,C 180,E1 -23348.199,E2 -23348.199} C_VEL
LIN {X 0,Y 183.657,Z 675.866,A -85,B 0,C 180,E1 -23352.046,E2 -23352.046} C_VEL
LIN {X 0,Y 188.229,Z 668.597,A -85,B 0,C 180,E1 -23355.192,E2 -23355.192} C_VEL
LIN {X 0,Y 189.438,Z 666.52,A -85,B 0,C 180,E1 -23355.966,E2 -23355.966} C_VEL
LIN {X 0,Y 189.466,Z 664.806,A -85,B 0,C 180,E1 -23356.85,E2 -23356.85} C_VEL
LIN {X 0,Y 181.472,Z 666.403,A -85,B 0,C 180,E1 -23358.825,E2 -23358.825} C_VEL
LIN {X 0,Y 176.393,Z 667.107,A -85,B 0,C 180,E1 -23360.397,E2 -23360.397} C_VEL
LIN {X 0,Y 170.167,Z 667.528,A -85,B 0,C 180,E1 -23362.843,E2 -23362.843} C_VEL
LIN {X 0,Y 169.573,Z 667.66,A -85,B 0,C 180,E1 -23363.433,E2 -23363.433} C_VEL
LIN {X 0,Y 169.308,Z 669.083,A -85,B 0,C 180,E1 -23363.92,E2 -23363.92} C_VEL
LIN {X 0,Y 167.704,Z 683.128,A -85,B 0,C 180,E1 -23366.272,E2 -23366.272} C_VEL
LIN {X 0,Y 166.164,Z 695.004,A -85,B 0,C 180,E1 -23368.863,E2 -23368.863} C_VEL
LIN {X 0,Y 164.867,Z 705.457,A -85,B 0,C 180,E1 -23371.691,E2 -23371.691} C_VEL
LIN {X 0,Y 163.589,Z 715.937,A -85,B 0,C 180,E1 -23375.237,E2 -23375.237} C_VEL
LIN {X 0,Y 162.827,Z 723.748,A -85,B 0,C 180,E1 -23378.478,E2 -23378.478} C_VEL
LIN {X 0,Y 162.217,Z 731.396,A -85,B 0,C 180,E1 -23382.403,E2 -23382.403} C_VEL
LIN {X 0,Y 161.983,Z 737.253,A -85,B 0,C 180,E1 -23386.195,E2 -23386.195} C_VEL
LIN {X 0,Y 162.138,Z 741.902,A -85,B 0,C 180,E1 -23390.016,E2 -23390.016} C_VEL
LIN {X 0,Y 162.77,Z 745.064,A -85,B 0,C 180,E1 -23393.289,E2 -23393.289} C_VEL
LIN {X 0,Y 164.15,Z 748.072,A -85,B 0,C 180,E1 -23397.547,E2 -23397.547} C_VEL
LIN {X 0,Y 166.854,Z 750.111,A -85,B 0,C 180,E1 -23402.415,E2 -23402.415} C_VEL
LIN {X 0,Y 169.53,Z 750.597,A -85,B 0,C 180,E1 -23405.733,E2 -23405.733} C_VEL
LIN {X 0,Y 173.172,Z 750.244,A -85,B 0,C 180,E1 -23409.343,E2 -23409.343} C_VEL
LIN {X 0,Y 178.888,Z 748.417,A -85,B 0,C 180,E1 -23413.635,E2 -23413.635} C_VEL
LIN {X 0,Y 185.666,Z 744.924,A -85,B 0,C 180,E1 -23417.628,E2 -23417.628} C_VEL
LIN {X 0,Y 191.33,Z 741.203,A -85,B 0,C 180,E1 -23420.424,E2 -23420.424} C_VEL
LIN {X 0,Y 198.739,Z 735.401,A -85,B 0,C 180,E1 -23423.49,E2 -23423.49} C_VEL
LIN {X 0,Y 205.403,Z 729.267,A -85,B 0,C 180,E1 -23425.866,E2 -23425.866} C_VEL
LIN {X 0,Y 212.616,Z 721.515,A -85,B 0,C 180,E1 -23428.102,E2 -23428.102} C_VEL
LIN {X 0,Y 218.717,Z 714.068,A -85,B 0,C 180,E1 -23429.815,E2 -23429.815} C_VEL
LIN {X 0,Y 225.7,Z 704.173,A -85,B 0,C 180,E1 -23431.553,E2 -23431.553} C_VEL
LIN {X 0,Y 232.217,Z 693.279,A -85,B 0,C 180,E1 -23433.009,E2 -23433.009} C_VEL
LIN {X 0,Y 238.041,Z 681.589,A -85,B 0,C 180,E1 -23434.236,E2 -23434.236} C_VEL
LIN {X 0,Y 242.954,Z 669.186,A -85,B 0,C 180,E1 -23435.209,E2 -23435.209} C_VEL
LIN {X 0,Y 247.161,Z 655.596,A -85,B 0,C 180,E1 -23435.992,E2 -23435.992} C_VEL
LIN {X 0,Y 255.244,Z 620.075,A -85,B 0,C 180,E1 -23437.408,E2 -23437.408} C_VEL
LIN {X 0,Y 255.294,Z 619.758,A -85,B 0,C 180,E1 -23438.564,E2 -23438.564} C_VEL
LIN {X 0,Y 253.557,Z 627.703,A -85,B 0,C 180,E1 -23439.172,E2 -23439.172} C_VEL
LIN {X 0,Y 253.034,Z 630.038,A -85,B 0,C 180,E1 -23439.259,E2 -23439.259} C_VEL
LIN {X 0,Y 251.743,Z 635.79,A -85,B 0,C 180,E1 -23439.337,E2 -23439.337} C_VEL
LIN {X 0,Y 247.107,Z 654.925,A -85,B 0,C 180,E1 -23438.711,E2 -23438.711} C_VEL
LIN {X 0,Y 245.522,Z 660.578,A -85,B 0,C 180,E1 -23438.784,E2 -23438.784} C_VEL
LIN {X 0,Y 241.016,Z 673.848,A -85,B 0,C 180,E1 -23439.396,E2 -23439.396} C_VEL
LIN {X 0,Y 234.735,Z 688.02,A -85,B 0,C 180,E1 -23440.225,E2 -23440.225} C_VEL
LIN {X 0,Y 227.24,Z 701.642,A -85,B 0,C 180,E1 -23441.406,E2 -23441.406} C_VEL
LIN {X 0,Y 219.964,Z 712.684,A -85,B 0,C 180,E1 -23442.7,E2 -23442.7} C_VEL
LIN {X 0,Y 211.589,Z 723.472,A -85,B 0,C 180,E1 -23444.424,E2 -23444.424} C_VEL
LIN {X 0,Y 203.732,Z 732.376,A -85,B 0,C 180,E1 -23446.372,E2 -23446.372} C_VEL
LIN {X 0,Y 195.077,Z 740.806,A -85,B 0,C 180,E1 -23448.887,E2 -23448.887} C_VEL
LIN {X 0,Y 187,Z 747.722,A -85,B 0,C 180,E1 -23451.671,E2 -23451.671} C_VEL
LIN {X 0,Y 178.709,Z 753.784,A -85,B 0,C 180,E1 -23455.229,E2 -23455.229} C_VEL
LIN {X 0,Y 173.3,Z 757.291,A -85,B 0,C 180,E1 -23458.179,E2 -23458.179} C_VEL
LIN {X 0,Y 168.974,Z 759.622,A -85,B 0,C 180,E1 -23460.862,E2 -23460.862} C_VEL
LIN {X 0,Y 164.378,Z 761.792,A -85,B 0,C 180,E1 -23464.683,E2 -23464.683} C_VEL
LIN {X 0,Y 160.046,Z 763.069,A -85,B 0,C 180,E1 -23469.429,E2 -23469.429} C_VEL
LIN {X 0,Y 158.335,Z 763.163,A -85,B 0,C 180,E1 -23471.894,E2 -23471.894} C_VEL
LIN {X 0,Y 156.263,Z 762.334,A -85,B 0,C 180,E1 -23477,E2 -23477} C_VEL
LIN {X 0,Y 155.589,Z 760.108,A -85,B 0,C 180,E1 -23482.208,E2 -23482.208} C_VEL
LIN {X 0,Y 155.84,Z 757.381,A -85,B 0,C 180,E1 -23486.117,E2 -23486.117} C_VEL
LIN {X 0,Y 156.304,Z 755.055,A -85,B 0,C 180,E1 -23488.707,E2 -23488.707} C_VEL
LIN {X 0,Y 156.368,Z 752.072,A -85,B 0,C 180,E1 -23491.283,E2 -23491.283} C_VEL
LIN {X 0,Y 156.313,Z 746.313,A -85,B 0,C 180,E1 -23495.155,E2 -23495.155} C_VEL
LIN {X 0,Y 156.466,Z 739.428,A -85,B 0,C 180,E1 -23498.813,E2 -23498.813} C_VEL
LIN {X 0,Y 156.883,Z 731.336,A -85,B 0,C 180,E1 -23502.281,E2 -23502.281} C_VEL
LIN {X 0,Y 157.904,Z 721.063,A -85,B 0,C 180,E1 -23505.815,E2 -23505.815} C_VEL
LIN {X 0,Y 158.161,Z 718.148,A -85,B 0,C 180,E1 -23506.783,E2 -23506.783} C_VEL
LIN {X 0,Y 159.534,Z 710.409,A -85,B 0,C 180,E1 -23510.631,E2 -23510.631} C_VEL
LIN {X 0,Y 161.572,Z 701.889,A -85,B 0,C 180,E1 -23514.011,E2 -23514.011} C_VEL
LIN {X 0,Y 164.017,Z 692.064,A -85,B 0,C 180,E1 -23517.078,E2 -23517.078} C_VEL
LIN {X 0,Y 166.882,Z 681.402,A -85,B 0,C 180,E1 -23519.654,E2 -23519.654} C_VEL
LIN {X 0,Y 169.601,Z 669.469,A -85,B 0,C 180,E1 -23521.888,E2 -23521.888} C_VEL
LIN {X 0,Y 172.092,Z 656.716,A -85,B 0,C 180,E1 -23523.628,E2 -23523.628} C_VEL
LIN {X 0,Y 173.894,Z 643.699,A -85,B 0,C 180,E1 -23524.918,E2 -23524.918} C_VEL
LIN {X 0,Y 175.004,Z 630.685,A -85,B 0,C 180,E1 -23525.757,E2 -23525.757} C_VEL
LIN {X 0,Y 175.768,Z 611.893,A -85,B 0,C 180,E1 -23526.528,E2 -23526.528} C_VEL
LIN {X 0,Y 172.577,Z 551.819,A -85,B 0,C 180,E1 -23530.049,E2 -23530.049} C_VEL
LIN {X 0,Y 171.987,Z 546.059,A -85,B 0,C 180,E1 -23530.46,E2 -23530.46} C_VEL
LIN {X 0,Y 165.446,Z 529.396,A -85,B 0,C 180,E1 -23532.835,E2 -23532.835} C_VEL
LIN {X 0,Y 161.243,Z 519.977,A -85,B 0,C 180,E1 -23534.518,E2 -23534.518} C_VEL
LIN {X 0,Y 159.355,Z 512.466,A -85,B 0,C 180,E1 -23538.581,E2 -23538.581} C_VEL
LIN {X 0,Y 157.255,Z 504.969,A -85,B 0,C 180,E1 -23543.253,E2 -23543.253} C_VEL
LIN {X 0,Y 157.283,Z 504.894,A -85,B 0,C 180,E1 -23548.093,E2 -23548.093} C_VEL
LIN {X 0,Y 157.311,Z 504.865,A -85,B 0,C 180,E1 -23553.463,E2 -23553.463} C_VEL
LIN {X 0,Y 157.383,Z 504.855,A -85,B 0,C 180,E1 -23559.665,E2 -23559.665} C_VEL
LIN {X 0,Y 157.467,Z 504.871,A -85,B 0,C 180,E1 -23564.466,E2 -23564.466} C_VEL
LIN {X 0,Y 157.717,Z 504.808,A -85,B 0,C 180,E1 -23569.732,E2 -23569.732} C_VEL
LIN {X 0,Y 157.799,Z 504.823,A -85,B 0,C 180,E1 -23572.321,E2 -23572.321} C_VEL
LIN {X 0,Y 158.245,Z 504.741,A -85,B 0,C 180,E1 -23579.999,E2 -23579.999} C_VEL
LIN {X 0,Y 157.772,Z 504.799,A -85,B 0,C 180,E1 -23587.679,E2 -23587.679} C_VEL
LIN {X 0,Y 157.668,Z 504.824,A -85,B 0,C 180,E1 -23591.316,E2 -23591.316} C_VEL
LIN {X 0,Y 157.466,Z 504.867,A -85,B 0,C 180,E1 -23595.532,E2 -23595.532} C_VEL
LIN {X 0,Y 157.358,Z 504.855,A -85,B 0,C 180,E1 -23600.933,E2 -23600.933} C_VEL
LIN {X 0,Y 157.302,Z 504.873,A -85,B 0,C 180,E1 -23606.686,E2 -23606.686} C_VEL
LIN {X 0,Y 157.264,Z 504.893,A -85,B 0,C 180,E1 -23612.429,E2 -23612.429} C_VEL
LIN {X 0,Y 157.257,Z 504.873,A -85,B 0,C 180,E1 -23616.452,E2 -23616.452} C_VEL
LIN {X 0,Y 157.219,Z 504.899,A -85,B 0,C 180,E1 -23622.107,E2 -23622.107} C_VEL
LIN {X 0,Y 157.262,Z 504.897,A -85,B 0,C 180,E1 -23627.912,E2 -23627.912} C_VEL
LIN {X 0,Y 157.316,Z 504.826,A -85,B 0,C 180,E1 -23633.526,E2 -23633.526} C_VEL
LIN {X 0,Y 157.376,Z 504.998,A -85,B 0,C 180,E1 -23639.475,E2 -23639.475} C_VEL
LIN {X 0,Y 157.611,Z 506.011,A -85,B 0,C 180,E1 -23640.071,E2 -23640.071} C_VEL
LIN {X 0,Y 159.208,Z 508.837,A -85,B 0,C 180,E1 -23640.752,E2 -23640.752} C_VEL
LIN {X 0,Y 160.68,Z 511.262,A -85,B 0,C 180,E1 -23641.31,E2 -23641.31} C_VEL
LIN {X 0,Y 167.01,Z 521.704,A -85,B 0,C 180,E1 -23643.536,E2 -23643.536} C_VEL
LIN {X 0,Y 175.328,Z 538.014,A -85,B 0,C 180,E1 -23646.261,E2 -23646.261} C_VEL
LIN {X 0,Y 178.348,Z 545.146,A -85,B 0,C 180,E1 -23647.226,E2 -23647.226} C_VEL
LIN {X 0,Y 177.032,Z 589.705,A -85,B 0,C 180,E1 -23649.114,E2 -23649.114} C_VEL
LIN {X 0,Y 176.141,Z 602.432,A -85,B 0,C 180,E1 -23650.042,E2 -23650.042} C_VEL
LIN {X 0,Y 174.851,Z 614.928,A -85,B 0,C 180,E1 -23651.399,E2 -23651.399} C_VEL
LIN {X 0,Y 172.983,Z 627.11,A -85,B 0,C 180,E1 -23653.178,E2 -23653.178} C_VEL
LIN {X 0,Y 170.716,Z 638.627,A -85,B 0,C 180,E1 -23655.399,E2 -23655.399} C_VEL
LIN {X 0,Y 168.394,Z 648.998,A -85,B 0,C 180,E1 -23657.959,E2 -23657.959} C_VEL
LIN {X 0,Y 166.038,Z 658.373,A -85,B 0,C 180,E1 -23660.871,E2 -23660.871} C_VEL
LIN {X 0,Y 163.611,Z 667.424,A -85,B 0,C 180,E1 -23664.458,E2 -23664.458} C_VEL
LIN {X 0,Y 161.772,Z 673.969,A -85,B 0,C 180,E1 -23667.697,E2 -23667.697} C_VEL
LIN {X 0,Y 160.184,Z 679.755,A -85,B 0,C 180,E1 -23671.261,E2 -23671.261} C_VEL
LIN {X 0,Y 159,Z 684.621,A -85,B 0,C 180,E1 -23675.076,E2 -23675.076} C_VEL
LIN {X 0,Y 158.323,Z 688.377,A -85,B 0,C 180,E1 -23678.942,E2 -23678.942} C_VEL
LIN {X 0,Y 158.15,Z 691.119,A -85,B 0,C 180,E1 -23682.842,E2 -23682.842} C_VEL
LIN {X 0,Y 158.308,Z 692.44,A -85,B 0,C 180,E1 -23685.452,E2 -23685.452} C_VEL
LIN {X 0,Y 158.728,Z 693.312,A -85,B 0,C 180,E1 -23688.06,E2 -23688.06} C_VEL
LIN {X 0,Y 160.339,Z 693.85,A -85,B 0,C 180,E1 -23693.238,E2 -23693.238} C_VEL
LIN {X 0,Y 161.543,Z 693.516,A -85,B 0,C 180,E1 -23695.793,E2 -23695.793} C_VEL
LIN {X 0,Y 162.986,Z 692.73,A -85,B 0,C 180,E1 -23698.32,E2 -23698.32} C_VEL
LIN {X 0,Y 165.445,Z 690.923,A -85,B 0,C 180,E1 -23701.835,E2 -23701.835} C_VEL
LIN {X 0,Y 168.791,Z 687.801,A -85,B 0,C 180,E1 -23705.661,E2 -23705.661} C_VEL
LIN {X 0,Y 172.813,Z 683.351,A -85,B 0,C 180,E1 -23709.405,E2 -23709.405} C_VEL
LIN {X 0,Y 177.529,Z 677.32,A -85,B 0,C 180,E1 -23713.075,E2 -23713.075} C_VEL
LIN {X 0,Y 181.547,Z 671.367,A -85,B 0,C 180,E1 -23715.829,E2 -23715.829} C_VEL
LIN {X 0,Y 181.466,Z 670.212,A -85,B 0,C 180,E1 -23716.573,E2 -23716.573} C_VEL
LIN {X 0,Y 172.212,Z 671.645,A -85,B 0,C 180,E1 -23719.236,E2 -23719.236} C_VEL
LIN {X 0,Y 167.468,Z 672.097,A -85,B 0,C 180,E1 -23720.988,E2 -23720.988} C_VEL
LIN {X 0,Y 163.209,Z 672.234,A -85,B 0,C 180,E1 -23722.926,E2 -23722.926} C_VEL
LIN {X 0,Y 162.07,Z 672.106,A -85,B 0,C 180,E1 -23723.785,E2 -23723.785} C_VEL
LIN {X 0,Y 161.756,Z 673.288,A -85,B 0,C 180,E1 -23724.376,E2 -23724.376} C_VEL
LIN {X 0,Y 160,Z 687.586,A -85,B 0,C 180,E1 -23727.133,E2 -23727.133} C_VEL
LIN {X 0,Y 158.626,Z 698.28,A -85,B 0,C 180,E1 -23729.738,E2 -23729.738} C_VEL
LIN {X 0,Y 157.234,Z 709.376,A -85,B 0,C 180,E1 -23733.093,E2 -23733.093} C_VEL
LIN {X 0,Y 156.153,Z 719.199,A -85,B 0,C 180,E1 -23736.809,E2 -23736.809} C_VEL
LIN {X 0,Y 155.351,Z 727.72,A -85,B 0,C 180,E1 -23740.854,E2 -23740.854} C_VEL
LIN {X 0,Y 155.035,Z 733.448,A -85,B 0,C 180,E1 -23744.218,E2 -23744.218} C_VEL
LIN {X 0,Y 154.951,Z 739.024,A -85,B 0,C 180,E1 -23748.224,E2 -23748.224} C_VEL
LIN {X 0,Y 155.403,Z 743.401,A -85,B 0,C 180,E1 -23752.203,E2 -23752.203} C_VEL
LIN {X 0,Y 156.081,Z 745.693,A -85,B 0,C 180,E1 -23754.834,E2 -23754.834} C_VEL
LIN {X 0,Y 158.121,Z 749.041,A -85,B 0,C 180,E1 -23760.001,E2 -23760.001} C_VEL
LIN {X 0,Y 159.633,Z 750.147,A -85,B 0,C 180,E1 -23762.524,E2 -23762.524} C_VEL
LIN {X 0,Y 163.658,Z 751.137,A -85,B 0,C 180,E1 -23767.403,E2 -23767.403} C_VEL
LIN {X 0,Y 168.869,Z 750.643,A -85,B 0,C 180,E1 -23772.011,E2 -23772.011} C_VEL
LIN {X 0,Y 175.308,Z 748.574,A -85,B 0,C 180,E1 -23776.298,E2 -23776.298} C_VEL
LIN {X 0,Y 182.752,Z 744.91,A -85,B 0,C 180,E1 -23780.25,E2 -23780.25} C_VEL
LIN {X 0,Y 188.961,Z 741.034,A -85,B 0,C 180,E1 -23782.988,E2 -23782.988} C_VEL
LIN {X 0,Y 195.712,Z 736.031,A -85,B 0,C 180,E1 -23785.527,E2 -23785.527} C_VEL
LIN {X 0,Y 204.097,Z 728.659,A -85,B 0,C 180,E1 -23788.261,E2 -23788.261} C_VEL
LIN {X 0,Y 211.989,Z 720.522,A -85,B 0,C 180,E1 -23790.456,E2 -23790.456} C_VEL
LIN {X 0,Y 219.791,Z 711.017,A -85,B 0,C 180,E1 -23792.385,E2 -23792.385} C_VEL
LIN {X 0,Y 226.755,Z 701.091,A -85,B 0,C 180,E1 -23793.911,E2 -23793.911} C_VEL
LIN {X 0,Y 233.68,Z 689.162,A -85,B 0,C 180,E1 -23795.293,E2 -23795.293} C_VEL
LIN {X 0,Y 238.969,Z 678.273,A -85,B 0,C 180,E1 -23796.29,E2 -23796.29} C_VEL
LIN {X 0,Y 243.783,Z 665.854,A -85,B 0,C 180,E1 -23797.129,E2 -23797.129} C_VEL
LIN {X 0,Y 247.376,Z 653.664,A -85,B 0,C 180,E1 -23797.748,E2 -23797.748} C_VEL
LIN {X 0,Y 249.632,Z 644.053,A -85,B 0,C 180,E1 -23798.156,E2 -23798.156} C_VEL
LIN {X 0,Y 245.522,Z 660.578,A -85,B 0,C 180,E1 -23798.784,E2 -23798.784} C_VEL
LIN {X 0,Y 243.652,Z 666.468,A -85,B 0,C 180,E1 -23798.882,E2 -23798.882} C_VEL
LIN {X 0,Y 239.93,Z 676.023,A -85,B 0,C 180,E1 -23798.643,E2 -23798.643} C_VEL
LIN {X 0,Y 235.639,Z 685.269,A -85,B 0,C 180,E1 -23798.452,E2 -23798.452} C_VEL
LIN {X 0,Y 232.87,Z 690.559,A -85,B 0,C 180,E1 -23798.63,E2 -23798.63} C_VEL
LIN {X 0,Y 225.898,Z 702.407,A -85,B 0,C 180,E1 -23799.641,E2 -23799.641} C_VEL
LIN {X 0,Y 216.897,Z 715.013,A -85,B 0,C 180,E1 -23801.114,E2 -23801.114} C_VEL
LIN {X 0,Y 208.279,Z 725.273,A -85,B 0,C 180,E1 -23802.78,E2 -23802.78} C_VEL
LIN {X 0,Y 198.822,Z 734.924,A -85,B 0,C 180,E1 -23805.007,E2 -23805.007} C_VEL
LIN {X 0,Y 191.167,Z 741.756,A -85,B 0,C 180,E1 -23807.142,E2 -23807.142} C_VEL
LIN {X 0,Y 183.881,Z 747.409,A -85,B 0,C 180,E1 -23809.473,E2 -23809.473} C_VEL
LIN {X 0,Y 177.179,Z 752.075,A -85,B 0,C 180,E1 -23812.057,E2 -23812.057} C_VEL
LIN {X 0,Y 171,Z 755.773,A -85,B 0,C 180,E1 -23814.868,E2 -23814.868} C_VEL
LIN {X 0,Y 163.759,Z 759.449,A -85,B 0,C 180,E1 -23818.998,E2 -23818.998} C_VEL
LIN {X 0,Y 157.972,Z 761.673,A -85,B 0,C 180,E1 -23823.579,E2 -23823.579} C_VEL
LIN {X 0,Y 153.415,Z 762.569,A -85,B 0,C 180,E1 -23828.497,E2 -23828.497} C_VEL
LIN {X 0,Y 150.341,Z 762.134,A -85,B 0,C 180,E1 -23833.706,E2 -23833.706} C_VEL
LIN {X 0,Y 148.809,Z 760.285,A -85,B 0,C 180,E1 -23839.106,E2 -23839.106} C_VEL
LIN {X 0,Y 148.76,Z 756.988,A -85,B 0,C 180,E1 -23844.574,E2 -23844.574} C_VEL
LIN {X 0,Y 149.409,Z 753.372,A -85,B 0,C 180,E1 -23848.648,E2 -23848.648} C_VEL
LIN {X 0,Y 149.43,Z 750.191,A -85,B 0,C 180,E1 -23851.343,E2 -23851.343} C_VEL
LIN {X 0,Y 149.375,Z 744.171,A -85,B 0,C 180,E1 -23855.395,E2 -23855.395} C_VEL
LIN {X 0,Y 149.553,Z 736.767,A -85,B 0,C 180,E1 -23859.292,E2 -23859.292} C_VEL
LIN {X 0,Y 150.09,Z 728.346,A -85,B 0,C 180,E1 -23862.846,E2 -23862.846} C_VEL
LIN {X 0,Y 150.97,Z 718.896,A -85,B 0,C 180,E1 -23866.214,E2 -23866.214} C_VEL
LIN {X 0,Y 152.221,Z 711.652,A -85,B 0,C 180,E1 -23870.255,E2 -23870.255} C_VEL
LIN {X 0,Y 154.383,Z 702.595,A -85,B 0,C 180,E1 -23874.182,E2 -23874.182} C_VEL
LIN {X 0,Y 157.1,Z 692.347,A -85,B 0,C 180,E1 -23877.649,E2 -23877.649} C_VEL
LIN {X 0,Y 159.99,Z 681.944,A -85,B 0,C 180,E1 -23880.337,E2 -23880.337} C_VEL
LIN {X 0,Y 162.817,Z 670.389,A -85,B 0,C 180,E1 -23882.649,E2 -23882.649} C_VEL
LIN {X 0,Y 165.341,Z 658.37,A -85,B 0,C 180,E1 -23884.457,E2 -23884.457} C_VEL
LIN {X 0,Y 167.325,Z 645.756,A -85,B 0,C 180,E1 -23885.826,E2 -23885.826} C_VEL
LIN {X 0,Y 168.665,Z 632.455,A -85,B 0,C 180,E1 -23886.813,E2 -23886.813} C_VEL
LIN {X 0,Y 169.624,Z 612.243,A -85,B 0,C 180,E1 -23887.698,E2 -23887.698} C_VEL
LIN {X 0,Y 166.558,Z 551.078,A -85,B 0,C 180,E1 -23891.44,E2 -23891.44} C_VEL
LIN {X 0,Y 166.156,Z 548.223,A -85,B 0,C 180,E1 -23891.683,E2 -23891.683} C_VEL
LIN {X 0,Y 160.322,Z 533.151,A -85,B 0,C 180,E1 -23893.962,E2 -23893.962} C_VEL
LIN {X 0,Y 155.265,Z 522.249,A -85,B 0,C 180,E1 -23896.009,E2 -23896.009} C_VEL
LIN {X 0,Y 153.702,Z 518.599,A -85,B 0,C 180,E1 -23896.805,E2 -23896.805} C_VEL
LIN {X 0,Y 151.691,Z 511.069,A -85,B 0,C 180,E1 -23901.284,E2 -23901.284} C_VEL
LIN {X 0,Y 150.234,Z 505.846,A -85,B 0,C 180,E1 -23904.83,E2 -23904.83} C_VEL
LIN {X 0,Y 150.197,Z 505.77,A -85,B 0,C 180,E1 -23909.021,E2 -23909.021} C_VEL
LIN {X 0,Y 150.233,Z 505.741,A -85,B 0,C 180,E1 -23912.716,E2 -23912.716} C_VEL
LIN {X 0,Y 150.34,Z 505.733,A -85,B 0,C 180,E1 -23919.205,E2 -23919.205} C_VEL
LIN {X 0,Y 150.372,Z 505.753,A -85,B 0,C 180,E1 -23923.713,E2 -23923.713} C_VEL
LIN {X 0,Y 150.64,Z 505.687,A -85,B 0,C 180,E1 -23929.244,E2 -23929.244} C_VEL
LIN {X 0,Y 150.733,Z 505.699,A -85,B 0,C 180,E1 -23931.958,E2 -23931.958} C_VEL
LIN {X 0,Y 151.206,Z 505.617,A -85,B 0,C 180,E1 -23939.999,E2 -23939.999} C_VEL
LIN {X 0,Y 150.712,Z 505.675,A -85,B 0,C 180,E1 -23948.041,E2 -23948.041} C_VEL
LIN {X 0,Y 150.598,Z 505.705,A -85,B 0,C 180,E1 -23951.501,E2 -23951.501} C_VEL
LIN {X 0,Y 150.37,Z 505.742,A -85,B 0,C 180,E1 -23956.285,E2 -23956.285} C_VEL
LIN {X 0,Y 150.339,Z 505.727,A -85,B 0,C 180,E1 -23960.793,E2 -23960.793} C_VEL
LIN {X 0,Y 150.232,Z 505.746,A -85,B 0,C 180,E1 -23967.283,E2 -23967.283} C_VEL
LIN {X 0,Y 150.204,Z 505.773,A -85,B 0,C 180,E1 -23972.634,E2 -23972.634} C_VEL
LIN {X 0,Y 150.162,Z 505.753,A -85,B 0,C 180,E1 -23977.475,E2 -23977.475} C_VEL
LIN {X 0,Y 150.155,Z 505.782,A -85,B 0,C 180,E1 -23981.514,E2 -23981.514} C_VEL
LIN {X 0,Y 150.182,Z 505.758,A -85,B 0,C 180,E1 -23985.423,E2 -23985.423} C_VEL
LIN {X 0,Y 150.214,Z 505.764,A -85,B 0,C 180,E1 -23989.086,E2 -23989.086} C_VEL
LIN {X 0,Y 150.229,Z 505.709,A -85,B 0,C 180,E1 -23992.681,E2 -23992.681} C_VEL
LIN {X 0,Y 150.257,Z 505.993,A -85,B 0,C 180,E1 -23997.408,E2 -23997.408} C_VEL
LIN {X 0,Y 150.521,Z 507.008,A -85,B 0,C 180,E1 -23997.925,E2 -23997.925} C_VEL
LIN {X 0,Y 152.166,Z 509.769,A -85,B 0,C 180,E1 -23998.669,E2 -23998.669} C_VEL
LIN {X 0,Y 153.234,Z 511.179,A -85,B 0,C 180,E1 -23999.099,E2 -23999.099} C_VEL
LIN {X 0,Y 159.84,Z 522.004,A -85,B 0,C 180,E1 -24001.684,E2 -24001.684} C_VEL
LIN {X 0,Y 165.388,Z 532.23,A -85,B 0,C 180,E1 -24003.691,E2 -24003.691} C_VEL
LIN {X 0,Y 170.698,Z 543.374,A -85,B 0,C 180,E1 -24005.517,E2 -24005.517} C_VEL
LIN {X 0,Y 172.395,Z 547.587,A -85,B 0,C 180,E1 -24006.101,E2 -24006.101} C_VEL
LIN {X 0,Y 171.025,Z 587.17,A -85,B 0,C 180,E1 -24007.778,E2 -24007.778} C_VEL
LIN {X 0,Y 170.201,Z 600.624,A -85,B 0,C 180,E1 -24008.665,E2 -24008.665} C_VEL
LIN {X 0,Y 168.966,Z 612.928,A -85,B 0,C 180,E1 -24009.935,E2 -24009.935} C_VEL
LIN {X 0,Y 167.192,Z 624.903,A -85,B 0,C 180,E1 -24011.628,E2 -24011.628} C_VEL
LIN {X 0,Y 164.786,Z 637.21,A -85,B 0,C 180,E1 -24013.91,E2 -24013.91} C_VEL
LIN {X 0,Y 162.305,Z 648.006,A -85,B 0,C 180,E1 -24016.546,E2 -24016.546} C_VEL
LIN {X 0,Y 159.988,Z 656.847,A -85,B 0,C 180,E1 -24019.244,E2 -24019.244} C_VEL
LIN {X 0,Y 157.371,Z 666.451,A -85,B 0,C 180,E1 -24022.95,E2 -24022.95} C_VEL
LIN {X 0,Y 155.176,Z 673.826,A -85,B 0,C 180,E1 -24026.574,E2 -24026.574} C_VEL
LIN {X 0,Y 153.583,Z 679.425,A -85,B 0,C 180,E1 -24030.004,E2 -24030.004} C_VEL
LIN {X 0,Y 152.206,Z 684.566,A -85,B 0,C 180,E1 -24033.976,E2 -24033.976} C_VEL
LIN {X 0,Y 151.368,Z 688.578,A -85,B 0,C 180,E1 -24038.011,E2 -24038.011} C_VEL
LIN {X 0,Y 151.096,Z 691.722,A -85,B 0,C 180,E1 -24042.374,E2 -24042.374} C_VEL
LIN {X 0,Y 151.366,Z 693.58,A -85,B 0,C 180,E1 -24046.18,E2 -24046.18} C_VEL
LIN {X 0,Y 152.661,Z 694.806,A -85,B 0,C 180,E1 -24051.615,E2 -24051.615} C_VEL
LIN {X 0,Y 153.697,Z 694.837,A -85,B 0,C 180,E1 -24054.306,E2 -24054.306} C_VEL
LIN {X 0,Y 155.031,Z 694.413,A -85,B 0,C 180,E1 -24056.962,E2 -24056.962} C_VEL
LIN {X 0,Y 156.617,Z 693.578,A -85,B 0,C 180,E1 -24059.583,E2 -24059.583} C_VEL
LIN {X 0,Y 159.062,Z 691.877,A -85,B 0,C 180,E1 -24062.915,E2 -24062.915} C_VEL
LIN {X 0,Y 162.915,Z 688.452,A -85,B 0,C 180,E1 -24067.158,E2 -24067.158} C_VEL
LIN {X 0,Y 166.868,Z 684.291,A -85,B 0,C 180,E1 -24070.704,E2 -24070.704} C_VEL
LIN {X 0,Y 171.457,Z 678.748,A -85,B 0,C 180,E1 -24074.178,E2 -24074.178} C_VEL
LIN {X 0,Y 173.047,Z 676.586,A -85,B 0,C 180,E1 -24075.3,E2 -24075.3} C_VEL
LIN {X 0,Y 173.125,Z 675.179,A -85,B 0,C 180,E1 -24076.362,E2 -24076.362} C_VEL
LIN {X 0,Y 163.091,Z 676.349,A -85,B 0,C 180,E1 -24079.731,E2 -24079.731} C_VEL
LIN {X 0,Y 158.745,Z 676.534,A -85,B 0,C 180,E1 -24081.699,E2 -24081.699} C_VEL
LIN {X 0,Y 154.62,Z 676.315,A -85,B 0,C 180,E1 -24084.164,E2 -24084.164} C_VEL
LIN {X 0,Y 154.216,Z 677.053,A -85,B 0,C 180,E1 -24084.831,E2 -24084.831} C_VEL
LIN {X 0,Y 152.219,Z 692.733,A -85,B 0,C 180,E1 -24088.32,E2 -24088.32} C_VEL
LIN {X 0,Y 150.783,Z 703.873,A -85,B 0,C 180,E1 -24091.462,E2 -24091.462} C_VEL
LIN {X 0,Y 149.54,Z 713.865,A -85,B 0,C 180,E1 -24094.978,E2 -24094.978} C_VEL
LIN {X 0,Y 148.728,Z 722.088,A -85,B 0,C 180,E1 -24098.518,E2 -24098.518} C_VEL
LIN {X 0,Y 148.143,Z 729.582,A -85,B 0,C 180,E1 -24102.482,E2 -24102.482} C_VEL
LIN {X 0,Y 147.891,Z 735.426,A -85,B 0,C 180,E1 -24106.256,E2 -24106.256} C_VEL
LIN {X 0,Y 148.055,Z 740.619,A -85,B 0,C 180,E1 -24110.437,E2 -24110.437} C_VEL
LIN {X 0,Y 148.907,Z 744.699,A -85,B 0,C 180,E1 -24114.585,E2 -24114.585} C_VEL
LIN {X 0,Y 150.898,Z 748.626,A -85,B 0,C 180,E1 -24120.001,E2 -24120.001} C_VEL
LIN {X 0,Y 154.292,Z 750.914,A -85,B 0,C 180,E1 -24125.228,E2 -24125.228} C_VEL
LIN {X 0,Y 159.007,Z 751.725,A -85,B 0,C 180,E1 -24130.184,E2 -24130.184} C_VEL
LIN {X 0,Y 161.847,Z 751.576,A -85,B 0,C 180,E1 -24132.541,E2 -24132.541} C_VEL
LIN {X 0,Y 168.465,Z 750.077,A -85,B 0,C 180,E1 -24136.98,E2 -24136.98} C_VEL
LIN {X 0,Y 176.122,Z 747.075,A -85,B 0,C 180,E1 -24141.048,E2 -24141.048} C_VEL
LIN {X 0,Y 182.501,Z 743.71,A -85,B 0,C 180,E1 -24143.851,E2 -24143.851} C_VEL
LIN {X 0,Y 191.864,Z 737.564,A -85,B 0,C 180,E1 -24147.251,E2 -24147.251} C_VEL
LIN {X 0,Y 199.354,Z 731.631,A -85,B 0,C 180,E1 -24149.575,E2 -24149.575} C_VEL
LIN {X 0,Y 207.807,Z 723.803,A -85,B 0,C 180,E1 -24151.815,E2 -24151.815} C_VEL
LIN {X 0,Y 215.593,Z 715.287,A -85,B 0,C 180,E1 -24153.655,E2 -24153.655} C_VEL
LIN {X 0,Y 223.724,Z 704.812,A -85,B 0,C 180,E1 -24155.343,E2 -24155.343} C_VEL
LIN {X 0,Y 231.21,Z 693.223,A -85,B 0,C 180,E1 -24156.733,E2 -24156.733} C_VEL
LIN {X 0,Y 237.262,Z 681.729,A -85,B 0,C 180,E1 -24157.797,E2 -24157.797} C_VEL
LIN {X 0,Y 236.4,Z 683.621,A -85,B 0,C 180,E1 -24158.201,E2 -24158.201} C_VEL
LIN {X 0,Y 232.87,Z 690.559,A -85,B 0,C 180,E1 -24158.63,E2 -24158.63} C_VEL
LIN {X 0,Y 229.968,Z 695.696,A -85,B 0,C 180,E1 -24158.845,E2 -24158.845} C_VEL
LIN {X 0,Y 224.518,Z 703.989,A -85,B 0,C 180,E1 -24158.849,E2 -24158.849} C_VEL
LIN {X 0,Y 218.611,Z 711.858,A -85,B 0,C 180,E1 -24158.95,E2 -24158.95} C_VEL
LIN {X 0,Y 215.004,Z 716.237,A -85,B 0,C 180,E1 -24159.33,E2 -24159.33} C_VEL
LIN {X 0,Y 206.602,Z 725.534,A -85,B 0,C 180,E1 -24160.806,E2 -24160.806} C_VEL
LIN {X 0,Y 197.349,Z 734.51,A -85,B 0,C 180,E1 -24162.785,E2 -24162.785} C_VEL
LIN {X 0,Y 188.72,Z 741.64,A -85,B 0,C 180,E1 -24164.958,E2 -24164.958} C_VEL
LIN {X 0,Y 178.625,Z 748.847,A -85,B 0,C 180,E1 -24168.016,E2 -24168.016} C_VEL
LIN {X 0,Y 169.489,Z 754.262,A -85,B 0,C 180,E1 -24171.534,E2 -24171.534} C_VEL
LIN {X 0,Y 165.287,Z 756.405,A -85,B 0,C 180,E1 -24173.463,E2 -24173.463} C_VEL
LIN {X 0,Y 157.733,Z 759.613,A -85,B 0,C 180,E1 -24177.673,E2 -24177.673} C_VEL
LIN {X 0,Y 151.635,Z 761.494,A -85,B 0,C 180,E1 -24182.383,E2 -24182.383} C_VEL
LIN {X 0,Y 146.831,Z 762.012,A -85,B 0,C 180,E1 -24187.481,E2 -24187.481} C_VEL
LIN {X 0,Y 143.55,Z 761.2,A -85,B 0,C 180,E1 -24192.913,E2 -24192.913} C_VEL
LIN {X 0,Y 141.926,Z 759.067,A -85,B 0,C 180,E1 -24198.571,E2 -24198.571} C_VEL
LIN {X 0,Y 141.767,Z 756.741,A -85,B 0,C 180,E1 -24202.526,E2 -24202.526} C_VEL
LIN {X 0,Y 142.249,Z 753.028,A -85,B 0,C 180,E1 -24207.163,E2 -24207.163} C_VEL
LIN {X 0,Y 142.589,Z 750.017,A -85,B 0,C 180,E1 -24209.995,E2 -24209.995} C_VEL
LIN {X 0,Y 142.484,Z 744.131,A -85,B 0,C 180,E1 -24214.238,E2 -24214.238} C_VEL
LIN {X 0,Y 142.55,Z 737.952,A -85,B 0,C 180,E1 -24217.786,E2 -24217.786} C_VEL
LIN {X 0,Y 142.864,Z 730.421,A -85,B 0,C 180,E1 -24221.344,E2 -24221.344} C_VEL
LIN {X 0,Y 143.813,Z 719.626,A -85,B 0,C 180,E1 -24225.587,E2 -24225.587} C_VEL
LIN {X 0,Y 144.919,Z 712.712,A -85,B 0,C 180,E1 -24229.84,E2 -24229.84} C_VEL
LIN {X 0,Y 146.963,Z 704.199,A -85,B 0,C 180,E1 -24233.979,E2 -24233.979} C_VEL
LIN {X 0,Y 149.601,Z 694.624,A -85,B 0,C 180,E1 -24237.596,E2 -24237.596} C_VEL
LIN {X 0,Y 152.76,Z 683.638,A -85,B 0,C 180,E1 -24240.78,E2 -24240.78} C_VEL
LIN {X 0,Y 155.646,Z 672.823,A -85,B 0,C 180,E1 -24243.189,E2 -24243.189} C_VEL
LIN {X 0,Y 158.418,Z 660.702,A -85,B 0,C 180,E1 -24245.215,E2 -24245.215} C_VEL
LIN {X 0,Y 160.49,Z 649.367,A -85,B 0,C 180,E1 -24246.625,E2 -24246.625} C_VEL
LIN {X 0,Y 162.239,Z 636.029,A -85,B 0,C 180,E1 -24247.797,E2 -24247.797} C_VEL
LIN {X 0,Y 163.267,Z 621.27,A -85,B 0,C 180,E1 -24248.564,E2 -24248.564} C_VEL
LIN {X 0,Y 163.508,Z 612.256,A -85,B 0,C 180,E1 -24248.974,E2 -24248.974} C_VEL
LIN {X 0,Y 160.775,Z 552.799,A -85,B 0,C 180,E1 -24252.767,E2 -24252.767} C_VEL
LIN {X 0,Y 160.342,Z 550.171,A -85,B 0,C 180,E1 -24253.022,E2 -24253.022} C_VEL
LIN {X 0,Y 154.611,Z 535.435,A -85,B 0,C 180,E1 -24255.433,E2 -24255.433} C_VEL
LIN {X 0,Y 150.457,Z 526.283,A -85,B 0,C 180,E1 -24257.252,E2 -24257.252} C_VEL
LIN {X 0,Y 147.756,Z 520.956,A -85,B 0,C 180,E1 -24258.475,E2 -24258.475} C_VEL
LIN {X 0,Y 146.061,Z 517.081,A -85,B 0,C 180,E1 -24259.491,E2 -24259.491} C_VEL
LIN {X 0,Y 144.094,Z 509.965,A -85,B 0,C 180,E1 -24264.176,E2 -24264.176} C_VEL
LIN {X 0,Y 143.161,Z 506.723,A -85,B 0,C 180,E1 -24266.664,E2 -24266.664} C_VEL
LIN {X 0,Y 143.18,Z 506.617,A -85,B 0,C 180,E1 -24272.061,E2 -24272.061} C_VEL
LIN {X 0,Y 143.266,Z 506.617,A -85,B 0,C 180,E1 -24278.743,E2 -24278.743} C_VEL
LIN {X 0,Y 143.306,Z 506.625,A -85,B 0,C 180,E1 -24282.886,E2 -24282.886} C_VEL
LIN {X 0,Y 143.583,Z 506.565,A -85,B 0,C 180,E1 -24288.708,E2 -24288.708} C_VEL
LIN {X 0,Y 143.653,Z 506.574,A -85,B 0,C 180,E1 -24291.559,E2 -24291.559} C_VEL
LIN {X 0,Y 144.164,Z 506.492,A -85,B 0,C 180,E1 -24299.999,E2 -24299.999} C_VEL
LIN {X 0,Y 143.636,Z 506.553,A -85,B 0,C 180,E1 -24308.44,E2 -24308.44} C_VEL
LIN {X 0,Y 143.536,Z 506.586,A -85,B 0,C 180,E1 -24311.713,E2 -24311.713} C_VEL
LIN {X 0,Y 143.304,Z 506.609,A -85,B 0,C 180,E1 -24317.112,E2 -24317.112} C_VEL
LIN {X 0,Y 143.265,Z 506.611,A -85,B 0,C 180,E1 -24321.255,E2 -24321.255} C_VEL
LIN {X 0,Y 143.178,Z 506.618,A -85,B 0,C 180,E1 -24327.938,E2 -24327.938} C_VEL
LIN {X 0,Y 143.153,Z 506.653,A -85,B 0,C 180,E1 -24333.435,E2 -24333.435} C_VEL
LIN {X 0,Y 143.057,Z 506.652,A -85,B 0,C 180,E1 -24339.69,E2 -24339.69} C_VEL
LIN {X 0,Y 143.095,Z 506.643,A -85,B 0,C 180,E1 -24343.439,E2 -24343.439} C_VEL
LIN {X 0,Y 143.127,Z 506.655,A -85,B 0,C 180,E1 -24347.437,E2 -24347.437} C_VEL
LIN {X 0,Y 143.129,Z 506.598,A -85,B 0,C 180,E1 -24351.778,E2 -24351.778} C_VEL
LIN {X 0,Y 143.147,Z 506.84,A -85,B 0,C 180,E1 -24354.812,E2 -24354.812} C_VEL
LIN {X 0,Y 143.433,Z 507.954,A -85,B 0,C 180,E1 -24355.47,E2 -24355.47} C_VEL
LIN {X 0,Y 145.25,Z 510.857,A -85,B 0,C 180,E1 -24356.38,E2 -24356.38} C_VEL
LIN {X 0,Y 146.314,Z 512.215,A -85,B 0,C 180,E1 -24356.85,E2 -24356.85} C_VEL
LIN {X 0,Y 151.249,Z 519.828,A -85,B 0,C 180,E1 -24359.002,E2 -24359.002} C_VEL
LIN {X 0,Y 158.15,Z 531.85,A -85,B 0,C 180,E1 -24361.773,E2 -24361.773} C_VEL
LIN {X 0,Y 164.959,Z 545.876,A -85,B 0,C 180,E1 -24364.308,E2 -24364.308} C_VEL
LIN {X 0,Y 166.268,Z 549.053,A -85,B 0,C 180,E1 -24364.788,E2 -24364.788} C_VEL
LIN {X 0,Y 164.851,Z 591.768,A -85,B 0,C 180,E1 -24366.735,E2 -24366.735} C_VEL
LIN {X 0,Y 163.868,Z 604.384,A -85,B 0,C 180,E1 -24367.715,E2 -24367.715} C_VEL
LIN {X 0,Y 162.312,Z 617.542,A -85,B 0,C 180,E1 -24369.241,E2 -24369.241} C_VEL
LIN {X 0,Y 160.236,Z 629.529,A -85,B 0,C 180,E1 -24371.132,E2 -24371.132} C_VEL
LIN {X 0,Y 157.762,Z 640.953,A -85,B 0,C 180,E1 -24373.506,E2 -24373.506} C_VEL
LIN {X 0,Y 155.187,Z 651.267,A -85,B 0,C 180,E1 -24376.25,E2 -24376.25} C_VEL
LIN {X 0,Y 152.579,Z 660.576,A -85,B 0,C 180,E1 -24379.387,E2 -24379.387} C_VEL
LIN {X 0,Y 149.923,Z 669.585,A -85,B 0,C 180,E1 -24383.274,E2 -24383.274} C_VEL
LIN {X 0,Y 147.681,Z 676.894,A -85,B 0,C 180,E1 -24387.277,E2 -24387.277} C_VEL
LIN {X 0,Y 145.953,Z 682.768,A -85,B 0,C 180,E1 -24391.384,E2 -24391.384} C_VEL
LIN {X 0,Y 144.774,Z 687.412,A -85,B 0,C 180,E1 -24395.576,E2 -24395.576} C_VEL
LIN {X 0,Y 144.168,Z 690.974,A -85,B 0,C 180,E1 -24399.829,E2 -24399.829} C_VEL
LIN {X 0,Y 144.129,Z 693.541,A -85,B 0,C 180,E1 -24404.116,E2 -24404.116} C_VEL
LIN {X 0,Y 144.428,Z 694.704,A -85,B 0,C 180,E1 -24406.98,E2 -24406.98} C_VEL
LIN {X 0,Y 145.951,Z 695.84,A -85,B 0,C 180,E1 -24412.663,E2 -24412.663} C_VEL
LIN {X 0,Y 147.105,Z 695.794,A -85,B 0,C 180,E1 -24415.471,E2 -24415.471} C_VEL
LIN {X 0,Y 150.316,Z 694.429,A -85,B 0,C 180,E1 -24420.956,E2 -24420.956} C_VEL
LIN {X 0,Y 152.691,Z 692.856,A -85,B 0,C 180,E1 -24424.057,E2 -24424.057} C_VEL
LIN {X 0,Y 157.174,Z 689.103,A -85,B 0,C 180,E1 -24428.761,E2 -24428.761} C_VEL
LIN {X 0,Y 161.742,Z 684.483,A -85,B 0,C 180,E1 -24432.658,E2 -24432.658} C_VEL
LIN {X 0,Y 164.441,Z 681.382,A -85,B 0,C 180,E1 -24434.678,E2 -24434.678} C_VEL
LIN {X 0,Y 165.213,Z 679.564,A -85,B 0,C 180,E1 -24436.038,E2 -24436.038} C_VEL
LIN {X 0,Y 158.65,Z 680.283,A -85,B 0,C 180,E1 -24438.359,E2 -24438.359} C_VEL
LIN {X 0,Y 154.185,Z 680.532,A -85,B 0,C 180,E1 -24440.348,E2 -24440.348} C_VEL
LIN {X 0,Y 147.252,Z 680.418,A -85,B 0,C 180,E1 -24444.488,E2 -24444.488} C_VEL
LIN {X 0,Y 146.745,Z 680.514,A -85,B 0,C 180,E1 -24445.236,E2 -24445.236} C_VEL
LIN {X 0,Y 146.54,Z 681.495,A -85,B 0,C 180,E1 -24445.701,E2 -24445.701} C_VEL
LIN {X 0,Y 144.775,Z 694.819,A -85,B 0,C 180,E1 -24448.951,E2 -24448.951} C_VEL
LIN {X 0,Y 143.443,Z 705.382,A -85,B 0,C 180,E1 -24452.191,E2 -24452.191} C_VEL
LIN {X 0,Y 142.278,Z 715.337,A -85,B 0,C 180,E1 -24455.952,E2 -24455.952} C_VEL
LIN {X 0,Y 141.501,Z 723.321,A -85,B 0,C 180,E1 -24459.656,E2 -24459.656} C_VEL
LIN {X 0,Y 140.999,Z 731.069,A -85,B 0,C 180,E1 -24464.09,E2 -24464.09} C_VEL
LIN {X 0,Y 140.892,Z 737.211,A -85,B 0,C 180,E1 -24468.492,E2 -24468.492} C_VEL
LIN {X 0,Y 141.519,Z 742.628,A -85,B 0,C 180,E1 -24473.362,E2 -24473.362} C_VEL
LIN {X 0,Y 143.105,Z 746.992,A -85,B 0,C 180,E1 -24478.594,E2 -24478.594} C_VEL
LIN {X 0,Y 145.208,Z 749.566,A -85,B 0,C 180,E1 -24482.775,E2 -24482.775} C_VEL
LIN {X 0,Y 149.351,Z 751.671,A -85,B 0,C 180,E1 -24488.117,E2 -24488.117} C_VEL
LIN {X 0,Y 154.806,Z 752.3,A -85,B 0,C 180,E1 -24493.121,E2 -24493.121} C_VEL
LIN {X 0,Y 161.604,Z 751.385,A -85,B 0,C 180,E1 -24497.724,E2 -24497.724} C_VEL
LIN {X 0,Y 169.492,Z 749.016,A -85,B 0,C 180,E1 -24501.913,E2 -24501.913} C_VEL
LIN {X 0,Y 178.38,Z 744.977,A -85,B 0,C 180,E1 -24505.684,E2 -24505.684} C_VEL
LIN {X 0,Y 185.685,Z 740.789,A -85,B 0,C 180,E1 -24508.237,E2 -24508.237} C_VEL
LIN {X 0,Y 194.718,Z 734.529,A -85,B 0,C 180,E1 -24510.953,E2 -24510.953} C_VEL
LIN {X 0,Y 202.838,Z 727.839,A -85,B 0,C 180,E1 -24513.011,E2 -24513.011} C_VEL
LIN {X 0,Y 211.479,Z 719.394,A -85,B 0,C 180,E1 -24514.979,E2 -24514.979} C_VEL
LIN {X 0,Y 219.873,Z 709.795,A -85,B 0,C 180,E1 -24516.637,E2 -24516.637} C_VEL
LIN {X 0,Y 224.993,Z 702.909,A -85,B 0,C 180,E1 -24517.55,E2 -24517.55} C_VEL
LIN {X 0,Y 224.156,Z 704.156,A -85,B 0,C 180,E1 -24517.946,E2 -24517.946} C_VEL
LIN {X 0,Y 215.539,Z 715.606,A -85,B 0,C 180,E1 -24519.244,E2 -24519.244} C_VEL
LIN {X 0,Y 215.004,Z 716.237,A -85,B 0,C 180,E1 -24519.33,E2 -24519.33} C_VEL
LIN {X 0,Y 212.4,Z 719.215,A -85,B 0,C 180,E1 -24519.555,E2 -24519.555} C_VEL
LIN {X 0,Y 202.64,Z 728.562,A -85,B 0,C 180,E1 -24519.483,E2 -24519.483} C_VEL
LIN {X 0,Y 199.807,Z 731.054,A -85,B 0,C 180,E1 -24519.811,E2 -24519.811} C_VEL
LIN {X 0,Y 189.345,Z 739.651,A -85,B 0,C 180,E1 -24522.063,E2 -24522.063} C_VEL
